LIN {X 0,Y 175.881,Z 377.344,A -85,B 0,C 180,E1 -22792.309,E2 -22792.309} C_VEL
LIN {X 0,Y 178.302,Z 371.488,A -85,B 0,C 180,E1 -22794.961,E2 -22794.961} C_VEL
LIN {X 0,Y 180.637,Z 365.547,A -85,B 0,C 180,E1 -22797.203,E2 -22797.203} C_VEL
LIN {X 0,Y 183.902,Z 356.997,A -85,B 0,C 180,E1 -22799.789,E2 -22799.789} C_VEL
LIN {X 0,Y 186.792,Z 348.822,A -85,B 0,C 180,E1 -22801.786,E2 -22801.786} C_VEL
LIN {X 0,Y 189.518,Z 340.315,A -85,B 0,C 180,E1 -22803.478,E2 -22803.478} C_VEL
LIN {X 0,Y 192.068,Z 331.606,A -85,B 0,C 180,E1 -22804.871,E2 -22804.871} C_VEL
LIN {X 0,Y 194.421,Z 321.851,A -85,B 0,C 180,E1 -22806.133,E2 -22806.133} C_VEL
LIN {X 0,Y 196.471,Z 311.774,A -85,B 0,C 180,E1 -22807.13,E2 -22807.13} C_VEL
LIN {X 0,Y 198.049,Z 301.956,A -85,B 0,C 180,E1 -22807.852,E2 -22807.852} C_VEL
LIN {X 0,Y 199.073,Z 292.344,A -85,B 0,C 180,E1 -22808.374,E2 -22808.374} C_VEL
LIN {X 0,Y 201.449,Z 250.434,A -85,B 0,C 180,E1 -22809.804,E2 -22809.804} C_VEL
LIN {X 0,Y 199.678,Z 238.962,A -85,B 0,C 180,E1 -22810.755,E2 -22810.755} C_VEL
LIN {X 0,Y 194.382,Z 225.961,A -85,B 0,C 180,E1 -22812.741,E2 -22812.741} C_VEL
LIN {X 0,Y 189.399,Z 215.335,A -85,B 0,C 180,E1 -22814.692,E2 -22814.692} C_VEL
LIN {X 0,Y 183.457,Z 204.391,A -85,B 0,C 180,E1 -22817.157,E2 -22817.157} C_VEL
LIN {X 0,Y 180.627,Z 199.673,A -85,B 0,C 180,E1 -22818.402,E2 -22818.402} C_VEL
LIN {X 0,Y 177.944,Z 195.27,A -85,B 0,C 180,E1 -22819.645,E2 -22819.645} C_VEL
LIN {X 0,Y 174.675,Z 190.219,A -85,B 0,C 180,E1 -22821.238,E2 -22821.238} C_VEL
LIN {X 0,Y 172.03,Z 186.816,A -85,B 0,C 180,E1 -22822.576,E2 -22822.576} C_VEL
LIN {X 0,Y 171.463,Z 185.167,A -85,B 0,C 180,E1 -22823.168,E2 -22823.168} C_VEL
LIN {X 0,Y 171.404,Z 184.674,A -85,B 0,C 180,E1 -22823.883,E2 -22823.883} C_VEL
LIN {X 0,Y 171.46,Z 184.628,A -85,B 0,C 180,E1 -22829.403,E2 -22829.403} C_VEL
LIN {X 0,Y 171.463,Z 184.591,A -85,B 0,C 180,E1 -22834.387,E2 -22834.387} C_VEL
LIN {X 0,Y 171.579,Z 184.562,A -85,B 0,C 180,E1 -22840.87,E2 -22840.87} C_VEL
LIN {X 0,Y 171.577,Z 184.609,A -85,B 0,C 180,E1 -22845.772,E2 -22845.772} C_VEL
LIN {X 0,Y 171.848,Z 184.523,A -85,B 0,C 180,E1 -22850.584,E2 -22850.584} C_VEL
LIN {X 0,Y 171.816,Z 184.583,A -85,B 0,C 180,E1 -22855.306,E2 -22855.306} C_VEL
LIN {X 0,Y 172.33,Z 184.463,A -85,B 0,C 180,E1 -22859.999,E2 -22859.999} C_VEL
LIN {X 0,Y 171.822,Z 184.581,A -85,B 0,C 180,E1 -22864.691,E2 -22864.691} C_VEL
LIN {X 0,Y 171.872,Z 184.523,A -85,B 0,C 180,E1 -22869.412,E2 -22869.412} C_VEL
LIN {X 0,Y 171.609,Z 184.608,A -85,B 0,C 180,E1 -22874.223,E2 -22874.223} C_VEL
LIN {X 0,Y 171.542,Z 184.57,A -85,B 0,C 180,E1 -22879.56,E2 -22879.56} C_VEL
LIN {X 0,Y 171.466,Z 184.596,A -85,B 0,C 180,E1 -22885.615,E2 -22885.615} C_VEL
LIN {X 0,Y 171.455,Z 184.624,A -85,B 0,C 180,E1 -22890.595,E2 -22890.595} C_VEL
LIN {X 0,Y 171.407,Z 184.674,A -85,B 0,C 180,E1 -22896.706,E2 -22896.706} C_VEL
LIN {X 0,Y 171.569,Z 185.534,A -85,B 0,C 180,E1 -22897.447,E2 -22897.447} C_VEL
LIN {X 0,Y 173.116,Z 188.45,A -85,B 0,C 180,E1 -22898.383,E2 -22898.383} C_VEL
LIN {X 0,Y 175.17,Z 190.413,A -85,B 0,C 180,E1 -22899.354,E2 -22899.354} C_VEL
LIN {X 0,Y 177.361,Z 193.784,A -85,B 0,C 180,E1 -22900.423,E2 -22900.423} C_VEL
LIN {X 0,Y 178.755,Z 195.514,A -85,B 0,C 180,E1 -22901.052,E2 -22901.052} C_VEL
LIN {X 0,Y 182.889,Z 201.427,A -85,B 0,C 180,E1 -22902.864,E2 -22902.864} C_VEL
LIN {X 0,Y 189.262,Z 210.902,A -85,B 0,C 180,E1 -22905.416,E2 -22905.416} C_VEL
LIN {X 0,Y 196.045,Z 222.621,A -85,B 0,C 180,E1 -22907.921,E2 -22907.921} C_VEL
LIN {X 0,Y 203.07,Z 236.728,A -85,B 0,C 180,E1 -22910.338,E2 -22910.338} C_VEL
LIN {X 0,Y 211.588,Z 254.961,A -85,B 0,C 180,E1 -22913.002,E2 -22913.002} C_VEL
LIN {X 0,Y 220.343,Z 269.518,A -85,B 0,C 180,E1 -22915.279,E2 -22915.279} C_VEL
LIN {X 0,Y 228.476,Z 280.884,A -85,B 0,C 180,E1 -22917.153,E2 -22917.153} C_VEL
LIN {X 0,Y 236.39,Z 290.633,A -85,B 0,C 180,E1 -22918.936,E2 -22918.936} C_VEL
LIN {X 0,Y 244.162,Z 299.37,A -85,B 0,C 180,E1 -22920.704,E2 -22920.704} C_VEL
LIN {X 0,Y 253.056,Z 308.497,A -85,B 0,C 180,E1 -22922.711,E2 -22922.711} C_VEL
LIN {X 0,Y 263.678,Z 317.89,A -85,B 0,C 180,E1 -22924.987,E2 -22924.987} C_VEL
LIN {X 0,Y 276.714,Z 327.934,A -85,B 0,C 180,E1 -22927.606,E2 -22927.606} C_VEL
LIN {X 0,Y 290.97,Z 338.137,A -85,B 0,C 180,E1 -22930.386,E2 -22930.386} C_VEL
LIN {X 0,Y 299.99,Z 344.721,A -85,B 0,C 180,E1 -22932.269,E2 -22932.269} C_VEL
LIN {X 0,Y 305.133,Z 348.259,A -85,B 0,C 180,E1 -22933.436,E2 -22933.436} C_VEL
LIN {X 0,Y 312.318,Z 353.434,A -85,B 0,C 180,E1 -22935.376,E2 -22935.376} C_VEL
LIN {X 0,Y 318.689,Z 357.408,A -85,B 0,C 180,E1 -22937.26,E2 -22937.26} C_VEL
LIN {X 0,Y 322.754,Z 360.096,A -85,B 0,C 180,E1 -22938.698,E2 -22938.698} C_VEL
LIN {X 0,Y 327.517,Z 363.396,A -85,B 0,C 180,E1 -22940.778,E2 -22940.778} C_VEL
LIN {X 0,Y 331.232,Z 365.579,A -85,B 0,C 180,E1 -22942.686,E2 -22942.686} C_VEL
LIN {X 0,Y 333.387,Z 366.65,A -85,B 0,C 180,E1 -22943.95,E2 -22943.95} C_VEL
LIN {X 0,Y 335.126,Z 367.434,A -85,B 0,C 180,E1 -22945.188,E2 -22945.188} C_VEL
LIN {X 0,Y 336.551,Z 367.967,A -85,B 0,C 180,E1 -22946.408,E2 -22946.408} C_VEL
LIN {X 0,Y 337.608,Z 368.387,A -85,B 0,C 180,E1 -22947.714,E2 -22947.714} C_VEL
LIN {X 0,Y 338.327,Z 368.639,A -85,B 0,C 180,E1 -22950,E2 -22950} C_VEL
LIN {X 0,Y 338.048,Z 368.614,A -85,B 0,C 180,E1 -22951.191,E2 -22951.191} C_VEL
LIN {X 0,Y 337.513,Z 368.349,A -85,B 0,C 180,E1 -22952.387,E2 -22952.387} C_VEL
LIN {X 0,Y 336.548,Z 367.946,A -85,B 0,C 180,E1 -22953.592,E2 -22953.592} C_VEL
LIN {X 0,Y 335.116,Z 367.413,A -85,B 0,C 180,E1 -22954.812,E2 -22954.812} C_VEL
LIN {X 0,Y 332.503,Z 366.264,A -85,B 0,C 180,E1 -22956.583,E2 -22956.583} C_VEL
LIN {X 0,Y 328.782,Z 364.143,A -85,B 0,C 180,E1 -22958.605,E2 -22958.605} C_VEL
LIN {X 0,Y 324.587,Z 361.397,A -85,B 0,C 180,E1 -22960.537,E2 -22960.537} C_VEL
LIN {X 0,Y 321.248,Z 359.031,A -85,B 0,C 180,E1 -22961.878,E2 -22961.878} C_VEL
LIN {X 0,Y 317.507,Z 356.675,A -85,B 0,C 180,E1 -22963.114,E2 -22963.114} C_VEL
LIN {X 0,Y 312.317,Z 353.442,A -85,B 0,C 180,E1 -22964.624,E2 -22964.624} C_VEL
LIN {X 0,Y 307.134,Z 349.761,A -85,B 0,C 180,E1 -22966.044,E2 -22966.044} C_VEL
LIN {X 0,Y 301.828,Z 346.015,A -85,B 0,C 180,E1 -22967.319,E2 -22967.319} C_VEL
LIN {X 0,Y 293.694,Z 340.243,A -85,B 0,C 180,E1 -22969.055,E2 -22969.055} C_VEL
LIN {X 0,Y 285.441,Z 334.313,A -85,B 0,C 180,E1 -22970.674,E2 -22970.674} C_VEL
LIN {X 0,Y 272.495,Z 324.875,A -85,B 0,C 180,E1 -22973.216,E2 -22973.216} C_VEL
LIN {X 0,Y 258.338,Z 313.345,A -85,B 0,C 180,E1 -22976.138,E2 -22976.138} C_VEL
LIN {X 0,Y 247.802,Z 303.312,A -85,B 0,C 180,E1 -22978.456,E2 -22978.456} C_VEL
LIN {X 0,Y 238.022,Z 292.543,A -85,B 0,C 180,E1 -22980.689,E2 -22980.689} C_VEL
LIN {X 0,Y 229.51,Z 282.137,A -85,B 0,C 180,E1 -22982.639,E2 -22982.639} C_VEL
LIN {X 0,Y 221.653,Z 271.453,A -85,B 0,C 180,E1 -22984.41,E2 -22984.41} C_VEL
LIN {X 0,Y 212.727,Z 256.998,A -85,B 0,C 180,E1 -22986.681,E2 -22986.681} C_VEL
LIN {X 0,Y 205.697,Z 242.652,A -85,B 0,C 180,E1 -22988.793,E2 -22988.793} C_VEL
LIN {X 0,Y 200.149,Z 230.678,A -85,B 0,C 180,E1 -22990.644,E2 -22990.644} C_VEL
LIN {X 0,Y 193.861,Z 218.632,A -85,B 0,C 180,E1 -22992.866,E2 -22992.866} C_VEL
LIN {X 0,Y 186.678,Z 206.839,A -85,B 0,C 180,E1 -22995.596,E2 -22995.596} C_VEL
LIN {X 0,Y 180.604,Z 198.174,A -85,B 0,C 180,E1 -22998.118,E2 -22998.118} C_VEL
LIN {X 0,Y 177.87,Z 194.262,A -85,B 0,C 180,E1 -22999.355,E2 -22999.355} C_VEL
LIN {X 0,Y 175.623,Z 191.34,A -85,B 0,C 180,E1 -23000.406,E2 -23000.406} C_VEL
LIN {X 0,Y 174.792,Z 189.863,A -85,B 0,C 180,E1 -23000.833,E2 -23000.833} C_VEL
LIN {X 0,Y 172.517,Z 187.642,A -85,B 0,C 180,E1 -23001.924,E2 -23001.924} C_VEL
LIN {X 0,Y 171.488,Z 185.196,A -85,B 0,C 180,E1 -23002.717,E2 -23002.717} C_VEL
LIN {X 0,Y 171.418,Z 184.641,A -85,B 0,C 180,E1 -23003.526,E2 -23003.526} C_VEL
LIN {X 0,Y 171.455,Z 184.624,A -85,B 0,C 180,E1 -23009.405,E2 -23009.405} C_VEL
LIN {X 0,Y 171.466,Z 184.596,A -85,B 0,C 180,E1 -23014.385,E2 -23014.385} C_VEL
LIN {X 0,Y 171.577,Z 184.565,A -85,B 0,C 180,E1 -23020.873,E2 -23020.873} C_VEL
LIN {X 0,Y 171.609,Z 184.608,A -85,B 0,C 180,E1 -23025.777,E2 -23025.777} C_VEL
LIN {X 0,Y 171.872,Z 184.523,A -85,B 0,C 180,E1 -23030.588,E2 -23030.588} C_VEL
LIN {X 0,Y 171.822,Z 184.581,A -85,B 0,C 180,E1 -23035.309,E2 -23035.309} C_VEL
LIN {X 0,Y 172.33,Z 184.463,A -85,B 0,C 180,E1 -23040.001,E2 -23040.001} C_VEL
LIN {X 0,Y 171.816,Z 184.583,A -85,B 0,C 180,E1 -23044.694,E2 -23044.694} C_VEL
LIN {X 0,Y 171.848,Z 184.523,A -85,B 0,C 180,E1 -23049.416,E2 -23049.416} C_VEL
LIN {X 0,Y 171.577,Z 184.609,A -85,B 0,C 180,E1 -23054.228,E2 -23054.228} C_VEL
LIN {X 0,Y 171.545,Z 184.568,A -85,B 0,C 180,E1 -23059.563,E2 -23059.563} C_VEL
LIN {X 0,Y 171.463,Z 184.591,A -85,B 0,C 180,E1 -23065.613,E2 -23065.613} C_VEL
LIN {X 0,Y 171.46,Z 184.628,A -85,B 0,C 180,E1 -23070.597,E2 -23070.597} C_VEL
LIN {X 0,Y 171.404,Z 184.741,A -85,B 0,C 180,E1 -23076.39,E2 -23076.39} C_VEL
LIN {X 0,Y 171.537,Z 185.46,A -85,B 0,C 180,E1 -23076.998,E2 -23076.998} C_VEL
LIN {X 0,Y 173.002,Z 188.32,A -85,B 0,C 180,E1 -23077.947,E2 -23077.947} C_VEL
LIN {X 0,Y 175.535,Z 191.428,A -85,B 0,C 180,E1 -23079.185,E2 -23079.185} C_VEL
LIN {X 0,Y 178.482,Z 195.95,A -85,B 0,C 180,E1 -23080.598,E2 -23080.598} C_VEL
LIN {X 0,Y 184.372,Z 205.931,A -85,B 0,C 180,E1 -23083.233,E2 -23083.233} C_VEL
LIN {X 0,Y 191.12,Z 218.728,A -85,B 0,C 180,E1 -23085.987,E2 -23085.987} C_VEL
LIN {X 0,Y 196.979,Z 232.036,A -85,B 0,C 180,E1 -23088.239,E2 -23088.239} C_VEL
LIN {X 0,Y 199.946,Z 239.938,A -85,B 0,C 180,E1 -23089.355,E2 -23089.355} C_VEL
LIN {X 0,Y 201.455,Z 251.296,A -85,B 0,C 180,E1 -23090.237,E2 -23090.237} C_VEL
LIN {X 0,Y 199.128,Z 292.429,A -85,B 0,C 180,E1 -23091.639,E2 -23091.639} C_VEL
LIN {X 0,Y 197.838,Z 303.708,A -85,B 0,C 180,E1 -23092.262,E2 -23092.262} C_VEL
LIN {X 0,Y 195.577,Z 316.798,A -85,B 0,C 180,E1 -23093.315,E2 -23093.315} C_VEL
LIN {X 0,Y 192.881,Z 328.342,A -85,B 0,C 180,E1 -23094.66,E2 -23094.66} C_VEL
LIN {X 0,Y 190.404,Z 337.616,A -85,B 0,C 180,E1 -23096.064,E2 -23096.064} C_VEL
LIN {X 0,Y 187.564,Z 346.555,A -85,B 0,C 180,E1 -23097.728,E2 -23097.728} C_VEL
LIN {X 0,Y 184.594,Z 355.079,A -85,B 0,C 180,E1 -23099.705,E2 -23099.705} C_VEL
LIN {X 0,Y 181.875,Z 362.294,A -85,B 0,C 180,E1 -23101.747,E2 -23101.747} C_VEL
LIN {X 0,Y 179.441,Z 368.494,A -85,B 0,C 180,E1 -23103.857,E2 -23103.857} C_VEL
LIN {X 0,Y 176.891,Z 375.034,A -85,B 0,C 180,E1 -23106.59,E2 -23106.59} C_VEL
LIN {X 0,Y 174.916,Z 379.533,A -85,B 0,C 180,E1 -23108.801,E2 -23108.801} C_VEL
LIN {X 0,Y 172.575,Z 385.026,A -85,B 0,C 180,E1 -23112.216,E2 -23112.216} C_VEL
LIN {X 0,Y 170.804,Z 389.353,A -85,B 0,C 180,E1 -23115.707,E2 -23115.707} C_VEL
LIN {X 0,Y 170.014,Z 391.725,A -85,B 0,C 180,E1 -23118.072,E2 -23118.072} C_VEL
LIN {X 0,Y 169.417,Z 393.528,A -85,B 0,C 180,E1 -23120.449,E2 -23120.449} C_VEL
LIN {X 0,Y 168.933,Z 395.987,A -85,B 0,C 180,E1 -23125.227,E2 -23125.227} C_VEL
LIN {X 0,Y 168.87,Z 396.632,A -85,B 0,C 180,E1 -23128.403,E2 -23128.403} C_VEL
LIN {X 0,Y 168.968,Z 396.739,A -85,B 0,C 180,E1 -23130,E2 -23130} C_VEL
LIN {X 0,Y 168.853,Z 396.52,A -85,B 0,C 180,E1 -23132.627,E2 -23132.627} C_VEL
LIN {X 0,Y 168.863,Z 395.985,A -85,B 0,C 180,E1 -23134.775,E2 -23134.775} C_VEL
LIN {X 0,Y 169.206,Z 394.079,A -85,B 0,C 180,E1 -23138.609,E2 -23138.609} C_VEL
LIN {X 0,Y 168.94,Z 392.807,A -85,B 0,C 180,E1 -23140.562,E2 -23140.562} C_VEL
LIN {X 0,Y 167.039,Z 390.176,A -85,B 0,C 180,E1 -23143.759,E2 -23143.759} C_VEL
LIN {X 0,Y 165.574,Z 386.861,A -85,B 0,C 180,E1 -23146.944,E2 -23146.944} C_VEL
LIN {X 0,Y 165.991,Z 384.451,A -85,B 0,C 180,E1 -23148.809,E2 -23148.809} C_VEL
LIN {X 0,Y 168.795,Z 378.306,A -85,B 0,C 180,E1 -23152.652,E2 -23152.652} C_VEL
LIN {X 0,Y 171.612,Z 371.914,A -85,B 0,C 180,E1 -23155.712,E2 -23155.712} C_VEL
LIN {X 0,Y 174.324,Z 365.355,A -85,B 0,C 180,E1 -23158.275,E2 -23158.275} C_VEL
LIN {X 0,Y 177.77,Z 356.805,A -85,B 0,C 180,E1 -23160.927,E2 -23160.927} C_VEL
LIN {X 0,Y 180.789,Z 348.631,A -85,B 0,C 180,E1 -23162.972,E2 -23162.972} C_VEL
LIN {X 0,Y 183.635,Z 340.123,A -85,B 0,C 180,E1 -23164.7,E2 -23164.7} C_VEL
LIN {X 0,Y 186.275,Z 331.414,A -85,B 0,C 180,E1 -23166.122,E2 -23166.122} C_VEL
LIN {X 0,Y 188.748,Z 321.66,A -85,B 0,C 180,E1 -23167.401,E2 -23167.401} C_VEL
LIN {X 0,Y 190.873,Z 311.583,A -85,B 0,C 180,E1 -23168.414,E2 -23168.414} C_VEL
LIN {X 0,Y 192.584,Z 301.13,A -85,B 0,C 180,E1 -23169.188,E2 -23169.188} C_VEL
LIN {X 0,Y 193.649,Z 291.081,A -85,B 0,C 180,E1 -23169.724,E2 -23169.724} C_VEL
LIN {X 0,Y 195.927,Z 251.075,A -85,B 0,C 180,E1 -23171.123,E2 -23171.123} C_VEL
LIN {X 0,Y 194.532,Z 241.871,A -85,B 0,C 180,E1 -23171.925,E2 -23171.925} C_VEL
LIN {X 0,Y 189.455,Z 229.158,A -85,B 0,C 180,E1 -23173.96,E2 -23173.96} C_VEL
LIN {X 0,Y 184.476,Z 218.447,A -85,B 0,C 180,E1 -23176.044,E2 -23176.044} C_VEL
LIN {X 0,Y 177.787,Z 206.032,A -85,B 0,C 180,E1 -23179.053,E2 -23179.053} C_VEL
LIN {X 0,Y 174.086,Z 200.115,A -85,B 0,C 180,E1 -23180.843,E2 -23180.843} C_VEL
LIN {X 0,Y 171.293,Z 195.651,A -85,B 0,C 180,E1 -23182.294,E2 -23182.294} C_VEL
LIN {X 0,Y 168.602,Z 191.975,A -85,B 0,C 180,E1 -23183.743,E2 -23183.743} C_VEL
LIN {X 0,Y 167.935,Z 190.842,A -85,B 0,C 180,E1 -23184.132,E2 -23184.132} C_VEL
LIN {X 0,Y 165.524,Z 188.584,A -85,B 0,C 180,E1 -23185.463,E2 -23185.463} C_VEL
LIN {X 0,Y 164.436,Z 186.081,A -85,B 0,C 180,E1 -23186.42,E2 -23186.42} C_VEL
LIN {X 0,Y 164.372,Z 185.526,A -85,B 0,C 180,E1 -23187.272,E2 -23187.272} C_VEL
LIN {X 0,Y 164.341,Z 185.476,A -85,B 0,C 180,E1 -23191.938,E2 -23191.938} C_VEL
LIN {X 0,Y 164.411,Z 185.471,A -85,B 0,C 180,E1 -23194.692,E2 -23194.692} C_VEL
LIN {X 0,Y 164.485,Z 185.449,A -85,B 0,C 180,E1 -23200.05,E2 -23200.05} C_VEL
LIN {X 0,Y 164.524,Z 185.484,A -85,B 0,C 180,E1 -23205.148,E2 -23205.148} C_VEL
LIN {X 0,Y 164.767,Z 185.404,A -85,B 0,C 180,E1 -23210.175,E2 -23210.175} C_VEL
LIN {X 0,Y 164.831,Z 185.413,A -85,B 0,C 180,E1 -23212.65,E2 -23212.65} C_VEL
LIN {X 0,Y 165.047,Z 185.39,A -85,B 0,C 180,E1 -23217.558,E2 -23217.558} C_VEL
LIN {X 0,Y 165.292,Z 185.339,A -85,B 0,C 180,E1 -23219.999,E2 -23219.999} C_VEL
LIN {X 0,Y 164.772,Z 185.461,A -85,B 0,C 180,E1 -23224.892,E2 -23224.892} C_VEL
LIN {X 0,Y 164.846,Z 185.416,A -85,B 0,C 180,E1 -23227.347,E2 -23227.347} C_VEL
LIN {X 0,Y 164.749,Z 185.414,A -85,B 0,C 180,E1 -23231.145,E2 -23231.145} C_VEL
LIN {X 0,Y 164.502,Z 185.454,A -85,B 0,C 180,E1 -23237.4,E2 -23237.4} C_VEL
LIN {X 0,Y 164.471,Z 185.452,A -85,B 0,C 180,E1 -23239.988,E2 -23239.988} C_VEL
LIN {X 0,Y 164.391,Z 185.472,A -85,B 0,C 180,E1 -23246.133,E2 -23246.133} C_VEL
LIN {X 0,Y 164.385,Z 185.491,A -85,B 0,C 180,E1 -23252.377,E2 -23252.377} C_VEL
LIN {X 0,Y 164.377,Z 185.815,A -85,B 0,C 180,E1 -23253.766,E2 -23253.766} C_VEL
LIN {X 0,Y 164.763,Z 187.147,A -85,B 0,C 180,E1 -23254.405,E2 -23254.405} C_VEL
LIN {X 0,Y 166.409,Z 189.67,A -85,B 0,C 180,E1 -23255.434,E2 -23255.434} C_VEL
LIN {X 0,Y 168.275,Z 191.164,A -85,B 0,C 180,E1 -23256.429,E2 -23256.429} C_VEL
LIN {X 0,Y 170.195,Z 194.383,A -85,B 0,C 180,E1 -23257.522,E2 -23257.522} C_VEL
LIN {X 0,Y 172.038,Z 196.358,A -85,B 0,C 180,E1 -23258.45,E2 -23258.45} C_VEL
LIN {X 0,Y 174.59,Z 199.966,A -85,B 0,C 180,E1 -23259.729,E2 -23259.729} C_VEL
LIN {X 0,Y 180.932,Z 209.13,A -85,B 0,C 180,E1 -23262.634,E2 -23262.634} C_VEL
LIN {X 0,Y 186.915,Z 218.677,A -85,B 0,C 180,E1 -23265.113,E2 -23265.113} C_VEL
LIN {X 0,Y 192.735,Z 229.168,A -85,B 0,C 180,E1 -23267.347,E2 -23267.347} C_VEL
LIN {X 0,Y 199.084,Z 242.459,A -85,B 0,C 180,E1 -23269.641,E2 -23269.641} C_VEL
LIN {X 0,Y 206.912,Z 259.443,A -85,B 0,C 180,E1 -23272.207,E2 -23272.207} C_VEL
LIN {X 0,Y 215.763,Z 274.325,A -85,B 0,C 180,E1 -23274.619,E2 -23274.619} C_VEL
LIN {X 0,Y 223.821,Z 285.817,A -85,B 0,C 180,E1 -23276.619,E2 -23276.619} C_VEL
LIN {X 0,Y 233.409,Z 297.849,A -85,B 0,C 180,E1 -23279.043,E2 -23279.043} C_VEL
LIN {X 0,Y 242.631,Z 308.097,A -85,B 0,C 180,E1 -23281.355,E2 -23281.355} C_VEL
LIN {X 0,Y 252.683,Z 317.792,A -85,B 0,C 180,E1 -23283.762,E2 -23283.762} C_VEL
LIN {X 0,Y 265.457,Z 328.251,A -85,B 0,C 180,E1 -23286.602,E2 -23286.602} C_VEL
LIN {X 0,Y 278.514,Z 337.618,A -85,B 0,C 180,E1 -23289.312,E2 -23289.312} C_VEL
LIN {X 0,Y 289.061,Z 344.904,A -85,B 0,C 180,E1 -23291.478,E2 -23291.478} C_VEL
LIN {X 0,Y 298.801,Z 351.715,A -85,B 0,C 180,E1 -23293.606,E2 -23293.606} C_VEL
LIN {X 0,Y 305.375,Z 356.469,A -85,B 0,C 180,E1 -23295.336,E2 -23295.336} C_VEL
LIN {X 0,Y 310.985,Z 360.104,A -85,B 0,C 180,E1 -23296.939,E2 -23296.939} C_VEL
LIN {X 0,Y 315.669,Z 362.977,A -85,B 0,C 180,E1 -23298.441,E2 -23298.441} C_VEL
LIN {X 0,Y 320.632,Z 366.467,A -85,B 0,C 180,E1 -23300.522,E2 -23300.522} C_VEL
LIN {X 0,Y 325.665,Z 369.51,A -85,B 0,C 180,E1 -23303.067,E2 -23303.067} C_VEL
LIN {X 0,Y 328.828,Z 371.056,A -85,B 0,C 180,E1 -23305.096,E2 -23305.096} C_VEL
LIN {X 0,Y 330.816,Z 371.833,A -85,B 0,C 180,E1 -23306.833,E2 -23306.833} C_VEL
LIN {X 0,Y 331.953,Z 372.324,A -85,B 0,C 180,E1 -23308.787,E2 -23308.787} C_VEL
LIN {X 0,Y 332.278,Z 372.333,A -85,B 0,C 180,E1 -23310,E2 -23310} C_VEL
LIN {X 0,Y 331.969,Z 372.307,A -85,B 0,C 180,E1 -23311.213,E2 -23311.213} C_VEL
LIN {X 0,Y 330.821,Z 371.835,A -85,B 0,C 180,E1 -23313.181,E2 -23313.181} C_VEL
LIN {X 0,Y 328.814,Z 371.044,A -85,B 0,C 180,E1 -23314.904,E2 -23314.904} C_VEL
LIN {X 0,Y 325.665,Z 369.505,A -85,B 0,C 180,E1 -23316.933,E2 -23316.933} C_VEL
LIN {X 0,Y 322.114,Z 367.424,A -85,B 0,C 180,E1 -23318.785,E2 -23318.785} C_VEL
LIN {X 0,Y 319.119,Z 365.447,A -85,B 0,C 180,E1 -23320.148,E2 -23320.148} C_VEL
LIN {X 0,Y 315.63,Z 363.006,A -85,B 0,C 180,E1 -23321.56,E2 -23321.56} C_VEL
LIN {X 0,Y 310.431,Z 359.762,A -85,B 0,C 180,E1 -23323.224,E2 -23323.224} C_VEL
LIN {X 0,Y 305.19,Z 356.343,A -85,B 0,C 180,E1 -23324.722,E2 -23324.722} C_VEL
LIN {X 0,Y 298.734,Z 351.703,A -85,B 0,C 180,E1 -23326.398,E2 -23326.398} C_VEL
LIN {X 0,Y 291.766,Z 346.896,A -85,B 0,C 180,E1 -23327.929,E2 -23327.929} C_VEL
LIN {X 0,Y 283.598,Z 341.056,A -85,B 0,C 180,E1 -23329.664,E2 -23329.664} C_VEL
LIN {X 0,Y 269.955,Z 331.548,A -85,B 0,C 180,E1 -23332.454,E2 -23332.454} C_VEL
LIN {X 0,Y 256.61,Z 321.192,A -85,B 0,C 180,E1 -23335.34,E2 -23335.34} C_VEL
LIN {X 0,Y 246.207,Z 311.766,A -85,B 0,C 180,E1 -23337.763,E2 -23337.763} C_VEL
LIN {X 0,Y 236.022,Z 300.893,A -85,B 0,C 180,E1 -23340.287,E2 -23340.287} C_VEL
LIN {X 0,Y 227.311,Z 290.369,A -85,B 0,C 180,E1 -23342.493,E2 -23342.493} C_VEL
LIN {X 0,Y 219.314,Z 279.593,A -85,B 0,C 180,E1 -23344.498,E2 -23344.498} C_VEL
LIN {X 0,Y 210.189,Z 265.266,A -85,B 0,C 180,E1 -23346.855,E2 -23346.855} C_VEL
LIN {X 0,Y 202.831,Z 251.158,A -85,B 0,C 180,E1 -23349.069,E2 -23349.069} C_VEL
LIN {X 0,Y 196.148,Z 236.12,A -85,B 0,C 180,E1 -23351.401,E2 -23351.401} C_VEL
LIN {X 0,Y 189.843,Z 223.734,A -85,B 0,C 180,E1 -23353.746,E2 -23353.746} C_VEL
LIN {X 0,Y 182.773,Z 211.915,A -85,B 0,C 180,E1 -23356.583,E2 -23356.583} C_VEL
LIN {X 0,Y 176.942,Z 203.408,A -85,B 0,C 180,E1 -23359.147,E2 -23359.147} C_VEL
LIN {X 0,Y 174.22,Z 199.577,A -85,B 0,C 180,E1 -23360.444,E2 -23360.444} C_VEL
LIN {X 0,Y 171.417,Z 195.571,A -85,B 0,C 180,E1 -23361.867,E2 -23361.867} C_VEL
LIN {X 0,Y 169.147,Z 192.916,A -85,B 0,C 180,E1 -23363.048,E2 -23363.048} C_VEL
LIN {X 0,Y 167.92,Z 190.819,A -85,B 0,C 180,E1 -23363.761,E2 -23363.761} C_VEL
LIN {X 0,Y 165.693,Z 188.828,A -85,B 0,C 180,E1 -23364.981,E2 -23364.981} C_VEL
LIN {X 0,Y 164.426,Z 186.04,A -85,B 0,C 180,E1 -23366.038,E2 -23366.038} C_VEL
LIN {X 0,Y 164.345,Z 185.511,A -85,B 0,C 180,E1 -23366.923,E2 -23366.923} C_VEL
LIN {X 0,Y 164.402,Z 185.506,A -85,B 0,C 180,E1 -23369.139,E2 -23369.139} C_VEL
LIN {X 0,Y 164.414,Z 185.477,A -85,B 0,C 180,E1 -23374.695,E2 -23374.695} C_VEL
LIN {X 0,Y 164.483,Z 185.45,A -85,B 0,C 180,E1 -23380.052,E2 -23380.052} C_VEL
LIN {X 0,Y 164.552,Z 185.488,A -85,B 0,C 180,E1 -23385.153,E2 -23385.153} C_VEL
LIN {X 0,Y 164.796,Z 185.403,A -85,B 0,C 180,E1 -23390.179,E2 -23390.179} C_VEL
LIN {X 0,Y 164.846,Z 185.416,A -85,B 0,C 180,E1 -23392.653,E2 -23392.653} C_VEL
LIN {X 0,Y 165.049,Z 185.385,A -85,B 0,C 180,E1 -23397.561,E2 -23397.561} C_VEL
LIN {X 0,Y 165.292,Z 185.339,A -85,B 0,C 180,E1 -23400.001,E2 -23400.001} C_VEL
LIN {X 0,Y 164.765,Z 185.462,A -85,B 0,C 180,E1 -23404.895,E2 -23404.895} C_VEL
LIN {X 0,Y 164.831,Z 185.413,A -85,B 0,C 180,E1 -23407.35,E2 -23407.35} C_VEL
LIN {X 0,Y 164.703,Z 185.419,A -85,B 0,C 180,E1 -23411.062,E2 -23411.062} C_VEL
LIN {X 0,Y 164.524,Z 185.484,A -85,B 0,C 180,E1 -23414.852,E2 -23414.852} C_VEL
LIN {X 0,Y 164.474,Z 185.451,A -85,B 0,C 180,E1 -23419.99,E2 -23419.99} C_VEL
LIN {X 0,Y 164.389,Z 185.468,A -85,B 0,C 180,E1 -23426.131,E2 -23426.131} C_VEL
LIN {X 0,Y 164.388,Z 185.5,A -85,B 0,C 180,E1 -23432.38,E2 -23432.38} C_VEL
LIN {X 0,Y 164.407,Z 185.864,A -85,B 0,C 180,E1 -23433.413,E2 -23433.413} C_VEL
LIN {X 0,Y 164.775,Z 187.218,A -85,B 0,C 180,E1 -23434.039,E2 -23434.039} C_VEL
LIN {X 0,Y 166.481,Z 189.733,A -85,B 0,C 180,E1 -23435.093,E2 -23435.093} C_VEL
LIN {X 0,Y 168.279,Z 191.289,A -85,B 0,C 180,E1 -23436.06,E2 -23436.06} C_VEL
LIN {X 0,Y 170.328,Z 194.545,A -85,B 0,C 180,E1 -23437.212,E2 -23437.212} C_VEL
LIN {X 0,Y 172.255,Z 197.096,A -85,B 0,C 180,E1 -23438.21,E2 -23438.21} C_VEL
LIN {X 0,Y 176.099,Z 203.374,A -85,B 0,C 180,E1 -23440.151,E2 -23440.151} C_VEL
LIN {X 0,Y 180.309,Z 210.544,A -85,B 0,C 180,E1 -23442.119,E2 -23442.119} C_VEL
LIN {X 0,Y 186.583,Z 222.723,A -85,B 0,C 180,E1 -23444.847,E2 -23444.847} C_VEL
LIN {X 0,Y 192.394,Z 236.231,A -85,B 0,C 180,E1 -23447.225,E2 -23447.225} C_VEL
LIN {X 0,Y 194.779,Z 242.867,A -85,B 0,C 180,E1 -23448.188,E2 -23448.188} C_VEL
LIN {X 0,Y 195.973,Z 251.524,A -85,B 0,C 180,E1 -23448.91,E2 -23448.91} C_VEL
LIN {X 0,Y 193.632,Z 292.079,A -85,B 0,C 180,E1 -23450.329,E2 -23450.329} C_VEL
LIN {X 0,Y 192.31,Z 303.337,A -85,B 0,C 180,E1 -23450.958,E2 -23450.958} C_VEL
LIN {X 0,Y 189.933,Z 316.607,A -85,B 0,C 180,E1 -23452.036,E2 -23452.036} C_VEL
LIN {X 0,Y 187.139,Z 328.151,A -85,B 0,C 180,E1 -23453.403,E2 -23453.403} C_VEL
LIN {X 0,Y 184.554,Z 337.424,A -85,B 0,C 180,E1 -23454.833,E2 -23454.833} C_VEL
LIN {X 0,Y 181.606,Z 346.363,A -85,B 0,C 180,E1 -23456.533,E2 -23456.533} C_VEL
LIN {X 0,Y 178.471,Z 354.886,A -85,B 0,C 180,E1 -23458.549,E2 -23458.549} C_VEL
LIN {X 0,Y 175.63,Z 362.102,A -85,B 0,C 180,E1 -23460.647,E2 -23460.647} C_VEL
LIN {X 0,Y 173.072,Z 368.302,A -85,B 0,C 180,E1 -23462.817,E2 -23462.817} C_VEL
LIN {X 0,Y 170.358,Z 374.842,A -85,B 0,C 180,E1 -23465.636,E2 -23465.636} C_VEL
LIN {X 0,Y 168.289,Z 379.341,A -85,B 0,C 180,E1 -23467.923,E2 -23467.923} C_VEL
LIN {X 0,Y 165.816,Z 384.834,A -85,B 0,C 180,E1 -23471.465,E2 -23471.465} C_VEL
LIN {X 0,Y 163.883,Z 389.16,A -85,B 0,C 180,E1 -23475.09,E2 -23475.09} C_VEL
LIN {X 0,Y 163.041,Z 391.532,A -85,B 0,C 180,E1 -23477.554,E2 -23477.554} C_VEL
LIN {X 0,Y 162.398,Z 393.336,A -85,B 0,C 180,E1 -23480.032,E2 -23480.032} C_VEL
LIN {X 0,Y 161.851,Z 395.795,A -85,B 0,C 180,E1 -23485.018,E2 -23485.018} C_VEL
LIN {X 0,Y 161.8,Z 396.389,A -85,B 0,C 180,E1 -23487.511,E2 -23487.511} C_VEL
LIN {X 0,Y 161.884,Z 396.548,A -85,B 0,C 180,E1 -23490,E2 -23490} C_VEL
LIN {X 0,Y 161.763,Z 396.388,A -85,B 0,C 180,E1 -23492.49,E2 -23492.49} C_VEL
LIN {X 0,Y 161.766,Z 395.793,A -85,B 0,C 180,E1 -23494.985,E2 -23494.985} C_VEL
LIN {X 0,Y 162.376,Z 393.335,A -85,B 0,C 180,E1 -23499.97,E2 -23499.97} C_VEL
LIN {X 0,Y 163.427,Z 390.379,A -85,B 0,C 180,E1 -23503.681,E2 -23503.681} C_VEL
LIN {X 0,Y 165.06,Z 386.386,A -85,B 0,C 180,E1 -23507.34,E2 -23507.34} C_VEL
LIN {X 0,Y 165.991,Z 384.451,A -85,B 0,C 180,E1 -23508.809,E2 -23508.809} C_VEL
LIN {X 0,Y 166.55,Z 381.856,A -85,B 0,C 180,E1 -23510.628,E2 -23510.628} C_VEL
LIN {X 0,Y 165.958,Z 377.196,A -85,B 0,C 180,E1 -23513.641,E2 -23513.641} C_VEL
LIN {X 0,Y 165.647,Z 372.04,A -85,B 0,C 180,E1 -23516.561,E2 -23516.561} C_VEL
LIN {X 0,Y 166.623,Z 368.424,A -85,B 0,C 180,E1 -23518.171,E2 -23518.171} C_VEL
LIN {X 0,Y 170.197,Z 360.284,A -85,B 0,C 180,E1 -23521.075,E2 -23521.075} C_VEL
LIN {X 0,Y 174.458,Z 349.573,A -85,B 0,C 180,E1 -23523.983,E2 -23523.983} C_VEL
LIN {X 0,Y 177.406,Z 341.283,A -85,B 0,C 180,E1 -23525.755,E2 -23525.755} C_VEL
LIN {X 0,Y 180.585,Z 331.222,A -85,B 0,C 180,E1 -23527.451,E2 -23527.451} C_VEL
LIN {X 0,Y 183.169,Z 321.469,A -85,B 0,C 180,E1 -23528.747,E2 -23528.747} C_VEL
LIN {X 0,Y 185.377,Z 311.392,A -85,B 0,C 180,E1 -23529.774,E2 -23529.774} C_VEL
LIN {X 0,Y 187.128,Z 300.987,A -85,B 0,C 180,E1 -23530.559,E2 -23530.559} C_VEL
LIN {X 0,Y 188.161,Z 291.748,A -85,B 0,C 180,E1 -23531.07,E2 -23531.07} C_VEL
LIN {X 0,Y 190.581,Z 252.189,A -85,B 0,C 180,E1 -23532.477,E2 -23532.477} C_VEL
LIN {X 0,Y 189.432,Z 244.667,A -85,B 0,C 180,E1 -23533.174,E2 -23533.174} C_VEL
LIN {X 0,Y 184.522,Z 232.205,A -85,B 0,C 180,E1 -23535.281,E2 -23535.281} C_VEL
LIN {X 0,Y 179.89,Z 222.208,A -85,B 0,C 180,E1 -23537.353,E2 -23537.353} C_VEL
LIN {X 0,Y 174.009,Z 211.003,A -85,B 0,C 180,E1 -23540.184,E2 -23540.184} C_VEL
LIN {X 0,Y 170.266,Z 204.841,A -85,B 0,C 180,E1 -23542.12,E2 -23542.12} C_VEL
LIN {X 0,Y 167.846,Z 200.943,A -85,B 0,C 180,E1 -23543.46,E2 -23543.46} C_VEL
LIN {X 0,Y 164.841,Z 196.752,A -85,B 0,C 180,E1 -23545.194,E2 -23545.194} C_VEL
LIN {X 0,Y 162.358,Z 193.942,A -85,B 0,C 180,E1 -23546.686,E2 -23546.686} C_VEL
LIN {X 0,Y 161.138,Z 191.822,A -85,B 0,C 180,E1 -23547.518,E2 -23547.518} C_VEL
LIN {X 0,Y 158.706,Z 189.741,A -85,B 0,C 180,E1 -23549.092,E2 -23549.092} C_VEL
LIN {X 0,Y 157.381,Z 186.949,A -85,B 0,C 180,E1 -23550.394,E2 -23550.394} C_VEL
LIN {X 0,Y 157.297,Z 186.405,A -85,B 0,C 180,E1 -23551.294,E2 -23551.294} C_VEL
LIN {X 0,Y 157.311,Z 186.378,A -85,B 0,C 180,E1 -23556.29,E2 -23556.29} C_VEL
LIN {X 0,Y 157.409,Z 186.325,A -85,B 0,C 180,E1 -23561.786,E2 -23561.786} C_VEL
LIN {X 0,Y 157.529,Z 186.336,A -85,B 0,C 180,E1 -23567.109,E2 -23567.109} C_VEL
LIN {X 0,Y 157.689,Z 186.286,A -85,B 0,C 180,E1 -23569.729,E2 -23569.729} C_VEL
LIN {X 0,Y 157.767,Z 186.287,A -85,B 0,C 180,E1 -23572.319,E2 -23572.319} C_VEL
LIN {X 0,Y 158.255,Z 186.214,A -85,B 0,C 180,E1 -23579.999,E2 -23579.999} C_VEL
LIN {X 0,Y 157.784,Z 186.29,A -85,B 0,C 180,E1 -23587.678,E2 -23587.678} C_VEL
LIN {X 0,Y 157.679,Z 186.294,A -85,B 0,C 180,E1 -23591.315,E2 -23591.315} C_VEL
LIN {X 0,Y 157.476,Z 186.357,A -85,B 0,C 180,E1 -23595.53,E2 -23595.53} C_VEL
LIN {X 0,Y 157.368,Z 186.344,A -85,B 0,C 180,E1 -23600.932,E2 -23600.932} C_VEL
LIN {X 0,Y 157.311,Z 186.35,A -85,B 0,C 180,E1 -23606.683,E2 -23606.683} C_VEL
LIN {X 0,Y 157.328,Z 186.674,A -85,B 0,C 180,E1 -23609.706,E2 -23609.706} C_VEL
LIN {X 0,Y 157.673,Z 187.862,A -85,B 0,C 180,E1 -23610.464,E2 -23610.464} C_VEL
LIN {X 0,Y 159.203,Z 190.362,A -85,B 0,C 180,E1 -23611.635,E2 -23611.635} C_VEL
LIN {X 0,Y 161.451,Z 192.096,A -85,B 0,C 180,E1 -23613.056,E2 -23613.056} C_VEL
LIN {X 0,Y 163.477,Z 195.455,A -85,B 0,C 180,E1 -23614.397,E2 -23614.397} C_VEL
LIN {X 0,Y 165.509,Z 197.573,A -85,B 0,C 180,E1 -23615.574,E2 -23615.574} C_VEL
LIN {X 0,Y 168.076,Z 201.156,A -85,B 0,C 180,E1 -23617.039,E2 -23617.039} C_VEL
LIN {X 0,Y 169.597,Z 203.288,A -85,B 0,C 180,E1 -23617.865,E2 -23617.865} C_VEL
LIN {X 0,Y 172.697,Z 207.657,A -85,B 0,C 180,E1 -23619.459,E2 -23619.459} C_VEL
LIN {X 0,Y 178.249,Z 215.949,A -85,B 0,C 180,E1 -23622.086,E2 -23622.086} C_VEL
LIN {X 0,Y 183.591,Z 224.799,A -85,B 0,C 180,E1 -23624.401,E2 -23624.401} C_VEL
LIN {X 0,Y 188.923,Z 234.749,A -85,B 0,C 180,E1 -23626.553,E2 -23626.553} C_VEL
LIN {X 0,Y 194.587,Z 247.049,A -85,B 0,C 180,E1 -23628.719,E2 -23628.719} C_VEL
LIN {X 0,Y 202.23,Z 263.839,A -85,B 0,C 180,E1 -23631.36,E2 -23631.36} C_VEL
LIN {X 0,Y 211.13,Z 279.041,A -85,B 0,C 180,E1 -23633.925,E2 -23633.925} C_VEL
LIN {X 0,Y 218.118,Z 289.426,A -85,B 0,C 180,E1 -23635.859,E2 -23635.859} C_VEL
LIN {X 0,Y 226.087,Z 299.905,A -85,B 0,C 180,E1 -23638.099,E2 -23638.099} C_VEL
LIN {X 0,Y 234.41,Z 309.57,A -85,B 0,C 180,E1 -23640.395,E2 -23640.395} C_VEL
LIN {X 0,Y 242.758,Z 318.279,A -85,B 0,C 180,E1 -23642.627,E2 -23642.627} C_VEL
LIN {X 0,Y 253.559,Z 327.7,A -85,B 0,C 180,E1 -23645.289,E2 -23645.289} C_VEL
LIN {X 0,Y 265.342,Z 336.567,A -85,B 0,C 180,E1 -23647.974,E2 -23647.974} C_VEL
LIN {X 0,Y 278.84,Z 345.674,A -85,B 0,C 180,E1 -23650.874,E2 -23650.874} C_VEL
LIN {X 0,Y 289.824,Z 353.121,A -85,B 0,C 180,E1 -23653.298,E2 -23653.298} C_VEL
LIN {X 0,Y 296.496,Z 357.754,A -85,B 0,C 180,E1 -23654.886,E2 -23654.886} C_VEL
LIN {X 0,Y 303.243,Z 362.435,A -85,B 0,C 180,E1 -23656.751,E2 -23656.751} C_VEL
LIN {X 0,Y 309.772,Z 366.471,A -85,B 0,C 180,E1 -23658.783,E2 -23658.783} C_VEL
LIN {X 0,Y 313.637,Z 369.208,A -85,B 0,C 180,E1 -23660.381,E2 -23660.381} C_VEL
LIN {X 0,Y 318.724,Z 372.421,A -85,B 0,C 180,E1 -23662.864,E2 -23662.864} C_VEL
LIN {X 0,Y 322.199,Z 374.133,A -85,B 0,C 180,E1 -23664.995,E2 -23664.995} C_VEL
LIN {X 0,Y 323.942,Z 374.862,A -85,B 0,C 180,E1 -23666.347,E2 -23666.347} C_VEL
LIN {X 0,Y 325.003,Z 375.291,A -85,B 0,C 180,E1 -23667.521,E2 -23667.521} C_VEL
LIN {X 0,Y 325.633,Z 375.574,A -85,B 0,C 180,E1 -23668.763,E2 -23668.763} C_VEL
LIN {X 0,Y 325.966,Z 375.601,A -85,B 0,C 180,E1 -23670,E2 -23670} C_VEL
LIN {X 0,Y 325.644,Z 375.562,A -85,B 0,C 180,E1 -23671.237,E2 -23671.237} C_VEL
LIN {X 0,Y 325.008,Z 375.279,A -85,B 0,C 180,E1 -23672.479,E2 -23672.479} C_VEL
LIN {X 0,Y 323.83,Z 374.817,A -85,B 0,C 180,E1 -23673.733,E2 -23673.733} C_VEL
LIN {X 0,Y 322.187,Z 374.133,A -85,B 0,C 180,E1 -23675.006,E2 -23675.006} C_VEL
LIN {X 0,Y 318.725,Z 372.388,A -85,B 0,C 180,E1 -23677.137,E2 -23677.137} C_VEL
LIN {X 0,Y 315.043,Z 370.158,A -85,B 0,C 180,E1 -23678.984,E2 -23678.984} C_VEL
LIN {X 0,Y 311.816,Z 367.97,A -85,B 0,C 180,E1 -23680.388,E2 -23680.388} C_VEL
LIN {X 0,Y 307.83,Z 365.284,A -85,B 0,C 180,E1 -23681.857,E2 -23681.857} C_VEL
LIN {X 0,Y 302.565,Z 361.993,A -85,B 0,C 180,E1 -23683.431,E2 -23683.431} C_VEL
LIN {X 0,Y 296.431,Z 357.74,A -85,B 0,C 180,E1 -23685.117,E2 -23685.117} C_VEL
LIN {X 0,Y 289.818,Z 353.141,A -85,B 0,C 180,E1 -23686.697,E2 -23686.697} C_VEL
LIN {X 0,Y 278.837,Z 345.675,A -85,B 0,C 180,E1 -23689.127,E2 -23689.127} C_VEL
LIN {X 0,Y 265.341,Z 336.573,A -85,B 0,C 180,E1 -23692.025,E2 -23692.025} C_VEL
LIN {X 0,Y 252.116,Z 326.576,A -85,B 0,C 180,E1 -23695.046,E2 -23695.046} C_VEL
LIN {X 0,Y 241.109,Z 316.705,A -85,B 0,C 180,E1 -23697.799,E2 -23697.799} C_VEL
LIN {X 0,Y 230.684,Z 305.429,A -85,B 0,C 180,E1 -23700.624,E2 -23700.624} C_VEL
LIN {X 0,Y 221.647,Z 294.174,A -85,B 0,C 180,E1 -23703.147,E2 -23703.147} C_VEL
LIN {X 0,Y 214.577,Z 284.271,A -85,B 0,C 180,E1 -23705.137,E2 -23705.137} C_VEL
LIN {X 0,Y 205.977,Z 270.615,A -85,B 0,C 180,E1 -23707.513,E2 -23707.513} C_VEL
LIN {X 0,Y 198.395,Z 255.928,A -85,B 0,C 180,E1 -23709.903,E2 -23709.903} C_VEL
LIN {X 0,Y 191.449,Z 240.113,A -85,B 0,C 180,E1 -23712.461,E2 -23712.461} C_VEL
LIN {X 0,Y 185.612,Z 228.344,A -85,B 0,C 180,E1 -23714.771,E2 -23714.771} C_VEL
LIN {X 0,Y 178.865,Z 216.851,A -85,B 0,C 180,E1 -23717.641,E2 -23717.641} C_VEL
LIN {X 0,Y 173.339,Z 208.611,A -85,B 0,C 180,E1 -23720.221,E2 -23720.221} C_VEL
LIN {X 0,Y 170.546,Z 204.641,A -85,B 0,C 180,E1 -23721.634,E2 -23721.634} C_VEL
LIN {X 0,Y 168.076,Z 201.16,A -85,B 0,C 180,E1 -23722.96,E2 -23722.96} C_VEL
LIN {X 0,Y 165.415,Z 197.403,A -85,B 0,C 180,E1 -23724.484,E2 -23724.484} C_VEL
LIN {X 0,Y 162.348,Z 193.895,A -85,B 0,C 180,E1 -23726.315,E2 -23726.315} C_VEL
LIN {X 0,Y 161.124,Z 191.81,A -85,B 0,C 180,E1 -23727.147,E2 -23727.147} C_VEL
LIN {X 0,Y 158.713,Z 189.779,A -85,B 0,C 180,E1 -23728.705,E2 -23728.705} C_VEL
LIN {X 0,Y 157.448,Z 187.137,A -85,B 0,C 180,E1 -23729.858,E2 -23729.858} C_VEL
LIN {X 0,Y 157.281,Z 186.434,A -85,B 0,C 180,E1 -23730.928,E2 -23730.928} C_VEL
LIN {X 0,Y 157.319,Z 186.35,A -85,B 0,C 180,E1 -23733.467,E2 -23733.467} C_VEL
LIN {X 0,Y 157.391,Z 186.335,A -85,B 0,C 180,E1 -23739.669,E2 -23739.669} C_VEL
LIN {X 0,Y 157.476,Z 186.357,A -85,B 0,C 180,E1 -23744.47,E2 -23744.47} C_VEL
LIN {X 0,Y 157.725,Z 186.283,A -85,B 0,C 180,E1 -23749.735,E2 -23749.735} C_VEL
LIN {X 0,Y 157.784,Z 186.29,A -85,B 0,C 180,E1 -23752.322,E2 -23752.322} C_VEL
LIN {X 0,Y 158.255,Z 186.214,A -85,B 0,C 180,E1 -23760.001,E2 -23760.001} C_VEL
LIN {X 0,Y 157.767,Z 186.287,A -85,B 0,C 180,E1 -23767.681,E2 -23767.681} C_VEL
LIN {X 0,Y 157.637,Z 186.299,A -85,B 0,C 180,E1 -23771.238,E2 -23771.238} C_VEL
LIN {X 0,Y 157.453,Z 186.349,A -85,B 0,C 180,E1 -23775.536,E2 -23775.536} C_VEL
LIN {X 0,Y 157.37,Z 186.344,A -85,B 0,C 180,E1 -23780.934,E2 -23780.934} C_VEL
LIN {X 0,Y 157.311,Z 186.347,A -85,B 0,C 180,E1 -23786.683,E2 -23786.683} C_VEL
LIN {X 0,Y 157.338,Z 186.67,A -85,B 0,C 180,E1 -23789.339,E2 -23789.339} C_VEL
LIN {X 0,Y 157.684,Z 187.891,A -85,B 0,C 180,E1 -23790.095,E2 -23790.095} C_VEL
LIN {X 0,Y 159.437,Z 190.578,A -85,B 0,C 180,E1 -23791.411,E2 -23791.411} C_VEL
LIN {X 0,Y 161.462,Z 192.14,A -85,B 0,C 180,E1 -23792.686,E2 -23792.686} C_VEL
LIN {X 0,Y 163.323,Z 195.264,A -85,B 0,C 180,E1 -23793.923,E2 -23793.923} C_VEL
LIN {X 0,Y 165.354,Z 197.322,A -85,B 0,C 180,E1 -23795.101,E2 -23795.101} C_VEL
LIN {X 0,Y 167.965,Z 201.07,A -85,B 0,C 180,E1 -23796.603,E2 -23796.603} C_VEL
LIN {X 0,Y 172.402,Z 208.345,A -85,B 0,C 180,E1 -23799.004,E2 -23799.004} C_VEL
LIN {X 0,Y 176.657,Z 215.861,A -85,B 0,C 180,E1 -23801.122,E2 -23801.122} C_VEL
LIN {X 0,Y 182.463,Z 227.449,A -85,B 0,C 180,E1 -23803.803,E2 -23803.803} C_VEL
LIN {X 0,Y 188.141,Z 241.145,A -85,B 0,C 180,E1 -23806.277,E2 -23806.277} C_VEL
LIN {X 0,Y 189.721,Z 245.736,A -85,B 0,C 180,E1 -23806.961,E2 -23806.961} C_VEL
LIN {X 0,Y 190.636,Z 252.792,A -85,B 0,C 180,E1 -23807.569,E2 -23807.569} C_VEL
LIN {X 0,Y 188.211,Z 291.894,A -85,B 0,C 180,E1 -23808.946,E2 -23808.946} C_VEL
LIN {X 0,Y 186.858,Z 303.06,A -85,B 0,C 180,E1 -23809.58,E2 -23809.58} C_VEL
LIN {X 0,Y 184.385,Z 316.415,A -85,B 0,C 180,E1 -23810.679,E2 -23810.679} C_VEL
LIN {X 0,Y 181.499,Z 327.96,A -85,B 0,C 180,E1 -23812.069,E2 -23812.069} C_VEL
LIN {X 0,Y 178.79,Z 337.232,A -85,B 0,C 180,E1 -23813.52,E2 -23813.52} C_VEL
LIN {X 0,Y 175.718,Z 346.171,A -85,B 0,C 180,E1 -23815.254,E2 -23815.254} C_VEL
LIN {X 0,Y 172.434,Z 354.694,A -85,B 0,C 180,E1 -23817.314,E2 -23817.314} C_VEL
LIN {X 0,Y 169.465,Z 361.91,A -85,B 0,C 180,E1 -23819.468,E2 -23819.468} C_VEL
LIN {X 0,Y 166.758,Z 368.109,A -85,B 0,C 180,E1 -23821.698,E2 -23821.698} C_VEL
LIN {X 0,Y 163.882,Z 374.649,A -85,B 0,C 180,E1 -23824.606,E2 -23824.606} C_VEL
LIN {X 0,Y 161.716,Z 379.149,A -85,B 0,C 180,E1 -23826.975,E2 -23826.975} C_VEL
LIN {X 0,Y 159.063,Z 384.641,A -85,B 0,C 180,E1 -23830.648,E2 -23830.648} C_VEL
LIN {X 0,Y 156.988,Z 388.967,A -85,B 0,C 180,E1 -23834.419,E2 -23834.419} C_VEL
LIN {X 0,Y 156.067,Z 391.339,A -85,B 0,C 180,E1 -23836.988,E2 -23836.988} C_VEL
LIN {X 0,Y 155.399,Z 393.144,A -85,B 0,C 180,E1 -23839.578,E2 -23839.578} C_VEL
LIN {X 0,Y 154.754,Z 395.603,A -85,B 0,C 180,E1 -23844.789,E2 -23844.789} C_VEL
LIN {X 0,Y 154.715,Z 396.318,A -85,B 0,C 180,E1 -23847.983,E2 -23847.983} C_VEL
LIN {X 0,Y 154.687,Z 396.348,A -85,B 0,C 180,E1 -23851.695,E2 -23851.695} C_VEL
LIN {X 0,Y 154.694,Z 395.601,A -85,B 0,C 180,E1 -23855.213,E2 -23855.213} C_VEL
LIN {X 0,Y 155.353,Z 393.143,A -85,B 0,C 180,E1 -23860.425,E2 -23860.425} C_VEL
LIN {X 0,Y 156.505,Z 390.187,A -85,B 0,C 180,E1 -23864.299,E2 -23864.299} C_VEL
LIN {X 0,Y 158.285,Z 386.194,A -85,B 0,C 180,E1 -23868.108,E2 -23868.108} C_VEL
LIN {X 0,Y 160.771,Z 381.065,A -85,B 0,C 180,E1 -23871.812,E2 -23871.812} C_VEL
LIN {X 0,Y 163.347,Z 375.805,A -85,B 0,C 180,E1 -23874.802,E2 -23874.802} C_VEL
LIN {X 0,Y 166.149,Z 369.486,A -85,B 0,C 180,E1 -23877.729,E2 -23877.729} C_VEL
LIN {X 0,Y 166.623,Z 368.424,A -85,B 0,C 180,E1 -23878.171,E2 -23878.171} C_VEL
LIN {X 0,Y 167.683,Z 364.736,A -85,B 0,C 180,E1 -23879.712,E2 -23879.712} C_VEL
LIN {X 0,Y 167.936,Z 358.33,A -85,B 0,C 180,E1 -23882.302,E2 -23882.302} C_VEL
LIN {X 0,Y 168.367,Z 351.444,A -85,B 0,C 180,E1 -23884.723,E2 -23884.723} C_VEL
LIN {X 0,Y 169.572,Z 346.855,A -85,B 0,C 180,E1 -23885.916,E2 -23885.916} C_VEL
LIN {X 0,Y 172.6,Z 338.389,A -85,B 0,C 180,E1 -23887.645,E2 -23887.645} C_VEL
LIN {X 0,Y 175.459,Z 329.399,A -85,B 0,C 180,E1 -23889.114,E2 -23889.114} C_VEL
LIN {X 0,Y 178.188,Z 319.264,A -85,B 0,C 180,E1 -23890.415,E2 -23890.415} C_VEL
LIN {X 0,Y 180.793,Z 307.213,A -85,B 0,C 180,E1 -23891.568,E2 -23891.568} C_VEL
LIN {X 0,Y 182.657,Z 293.895,A -85,B 0,C 180,E1 -23892.428,E2 -23892.428} C_VEL
LIN {X 0,Y 184.177,Z 273.194,A -85,B 0,C 180,E1 -23893.208,E2 -23893.208} C_VEL
LIN {X 0,Y 185.333,Z 253.46,A -85,B 0,C 180,E1 -23893.903,E2 -23893.903} C_VEL
LIN {X 0,Y 184.447,Z 247.467,A -85,B 0,C 180,E1 -23894.485,E2 -23894.485} C_VEL
LIN {X 0,Y 179.172,Z 233.936,A -85,B 0,C 180,E1 -23896.925,E2 -23896.925} C_VEL
LIN {X 0,Y 173.855,Z 222.782,A -85,B 0,C 180,E1 -23899.508,E2 -23899.508} C_VEL
LIN {X 0,Y 169.493,Z 214.598,A -85,B 0,C 180,E1 -23901.798,E2 -23901.798} C_VEL
LIN {X 0,Y 166.823,Z 210.024,A -85,B 0,C 180,E1 -23903.291,E2 -23903.291} C_VEL
LIN {X 0,Y 164.591,Z 206.365,A -85,B 0,C 180,E1 -23904.607,E2 -23904.607} C_VEL
LIN {X 0,Y 161.843,Z 202.546,A -85,B 0,C 180,E1 -23906.286,E2 -23906.286} C_VEL
LIN {X 0,Y 159.202,Z 199.126,A -85,B 0,C 180,E1 -23908.01,E2 -23908.01} C_VEL
LIN {X 0,Y 158.442,Z 198,A -85,B 0,C 180,E1 -23908.545,E2 -23908.545} C_VEL
LIN {X 0,Y 155.968,Z 195.419,A -85,B 0,C 180,E1 -23910.285,E2 -23910.285} C_VEL
LIN {X 0,Y 154.515,Z 192.925,A -85,B 0,C 180,E1 -23911.471,E2 -23911.471} C_VEL
LIN {X 0,Y 151.885,Z 190.885,A -85,B 0,C 180,E1 -23913.547,E2 -23913.547} C_VEL
LIN {X 0,Y 150.49,Z 188.476,A -85,B 0,C 180,E1 -23914.946,E2 -23914.946} C_VEL
LIN {X 0,Y 150.275,Z 187.492,A -85,B 0,C 180,E1 -23915.843,E2 -23915.843} C_VEL
LIN {X 0,Y 150.341,Z 187.205,A -85,B 0,C 180,E1 -23920.898,E2 -23920.898} C_VEL
LIN {X 0,Y 150.436,Z 187.23,A -85,B 0,C 180,E1 -23926.49,E2 -23926.49} C_VEL
LIN {X 0,Y 150.611,Z 187.169,A -85,B 0,C 180,E1 -23929.241,E2 -23929.241} C_VEL
LIN {X 0,Y 150.704,Z 187.161,A -85,B 0,C 180,E1 -23931.956,E2 -23931.956} C_VEL
LIN {X 0,Y 151.216,Z 187.09,A -85,B 0,C 180,E1 -23939.999,E2 -23939.999} C_VEL
LIN {X 0,Y 150.723,Z 187.163,A -85,B 0,C 180,E1 -23948.04,E2 -23948.04} C_VEL
LIN {X 0,Y 150.61,Z 187.175,A -85,B 0,C 180,E1 -23951.499,E2 -23951.499} C_VEL
LIN {X 0,Y 150.38,Z 187.225,A -85,B 0,C 180,E1 -23956.283,E2 -23956.283} C_VEL
LIN {X 0,Y 150.349,Z 187.215,A -85,B 0,C 180,E1 -23960.791,E2 -23960.791} C_VEL
LIN {X 0,Y 150.261,Z 187.493,A -85,B 0,C 180,E1 -23964.616,E2 -23964.616} C_VEL
LIN {X 0,Y 150.544,Z 188.595,A -85,B 0,C 180,E1 -23965.505,E2 -23965.505} C_VEL
LIN {X 0,Y 152.17,Z 191.253,A -85,B 0,C 180,E1 -23967.084,E2 -23967.084} C_VEL
LIN {X 0,Y 154.788,Z 193.216,A -85,B 0,C 180,E1 -23969.121,E2 -23969.121} C_VEL
LIN {X 0,Y 156.751,Z 196.485,A -85,B 0,C 180,E1 -23970.683,E2 -23970.683} C_VEL
LIN {X 0,Y 158.909,Z 198.503,A -85,B 0,C 180,E1 -23972.149,E2 -23972.149} C_VEL
LIN {X 0,Y 161.388,Z 202.115,A -85,B 0,C 180,E1 -23973.818,E2 -23973.818} C_VEL
LIN {X 0,Y 162.748,Z 203.677,A -85,B 0,C 180,E1 -23974.651,E2 -23974.651} C_VEL
LIN {X 0,Y 166.629,Z 209.198,A -85,B 0,C 180,E1 -23976.942,E2 -23976.942} C_VEL
LIN {X 0,Y 169.445,Z 213.265,A -85,B 0,C 180,E1 -23978.472,E2 -23978.472} C_VEL
LIN {X 0,Y 175.862,Z 223.093,A -85,B 0,C 180,E1 -23981.646,E2 -23981.646} C_VEL
LIN {X 0,Y 182.911,Z 235.738,A -85,B 0,C 180,E1 -23984.784,E2 -23984.784} C_VEL
LIN {X 0,Y 189.069,Z 249.077,A -85,B 0,C 180,E1 -23987.327,E2 -23987.327} C_VEL
LIN {X 0,Y 197.414,Z 267.895,A -85,B 0,C 180,E1 -23990.414,E2 -23990.414} C_VEL
LIN {X 0,Y 205.386,Z 282.038,A -85,B 0,C 180,E1 -23992.911,E2 -23992.911} C_VEL
LIN {X 0,Y 211.649,Z 291.914,A -85,B 0,C 180,E1 -23994.853,E2 -23994.853} C_VEL
LIN {X 0,Y 219.329,Z 302.582,A -85,B 0,C 180,E1 -23997.258,E2 -23997.258} C_VEL
LIN {X 0,Y 227.668,Z 312.732,A -85,B 0,C 180,E1 -23999.806,E2 -23999.806} C_VEL
LIN {X 0,Y 237.415,Z 322.956,A -85,B 0,C 180,E1 -24002.629,E2 -24002.629} C_VEL
LIN {X 0,Y 247.526,Z 331.769,A -85,B 0,C 180,E1 -24005.307,E2 -24005.307} C_VEL
LIN {X 0,Y 260.657,Z 341.432,A -85,B 0,C 180,E1 -24008.465,E2 -24008.465} C_VEL
LIN {X 0,Y 274.191,Z 350.188,A -85,B 0,C 180,E1 -24011.506,E2 -24011.506} C_VEL
LIN {X 0,Y 286.596,Z 358.156,A -85,B 0,C 180,E1 -24014.351,E2 -24014.351} C_VEL
LIN {X 0,Y 293.532,Z 362.975,A -85,B 0,C 180,E1 -24016.147,E2 -24016.147} C_VEL
LIN {X 0,Y 299.382,Z 366.841,A -85,B 0,C 180,E1 -24017.803,E2 -24017.803} C_VEL
LIN {X 0,Y 304.112,Z 369.804,A -85,B 0,C 180,E1 -24019.346,E2 -24019.346} C_VEL
LIN {X 0,Y 307.632,Z 372.245,A -85,B 0,C 180,E1 -24020.798,E2 -24020.798} C_VEL
LIN {X 0,Y 311.691,Z 374.869,A -85,B 0,C 180,E1 -24022.792,E2 -24022.792} C_VEL
LIN {X 0,Y 315.287,Z 376.744,A -85,B 0,C 180,E1 -24024.885,E2 -24024.885} C_VEL
LIN {X 0,Y 317.044,Z 377.489,A -85,B 0,C 180,E1 -24026.187,E2 -24026.187} C_VEL
LIN {X 0,Y 318.352,Z 377.992,A -85,B 0,C 180,E1 -24027.469,E2 -24027.469} C_VEL
LIN {X 0,Y 319.068,Z 378.311,A -85,B 0,C 180,E1 -24028.738,E2 -24028.738} C_VEL
LIN {X 0,Y 319.441,Z 378.367,A -85,B 0,C 180,E1 -24030,E2 -24030} C_VEL
LIN {X 0,Y 319.077,Z 378.305,A -85,B 0,C 180,E1 -24031.262,E2 -24031.262} C_VEL
LIN {X 0,Y 318.356,Z 377.988,A -85,B 0,C 180,E1 -24032.531,E2 -24032.531} C_VEL
LIN {X 0,Y 316.981,Z 377.457,A -85,B 0,C 180,E1 -24033.878,E2 -24033.878} C_VEL
LIN {X 0,Y 315.279,Z 376.748,A -85,B 0,C 180,E1 -24035.116,E2 -24035.116} C_VEL
LIN {X 0,Y 311.706,Z 374.809,A -85,B 0,C 180,E1 -24037.231,E2 -24037.231} C_VEL
LIN {X 0,Y 307.615,Z 372.232,A -85,B 0,C 180,E1 -24039.203,E2 -24039.203} C_VEL
LIN {X 0,Y 304.087,Z 369.798,A -85,B 0,C 180,E1 -24040.655,E2 -24040.655} C_VEL
LIN {X 0,Y 298.202,Z 366.129,A -85,B 0,C 180,E1 -24042.544,E2 -24042.544} C_VEL
LIN {X 0,Y 290.559,Z 360.891,A -85,B 0,C 180,E1 -24044.648,E2 -24044.648} C_VEL
LIN {X 0,Y 282.365,Z 355.532,A -85,B 0,C 180,E1 -24046.617,E2 -24046.617} C_VEL
LIN {X 0,Y 271.456,Z 348.509,A -85,B 0,C 180,E1 -24049.097,E2 -24049.097} C_VEL
LIN {X 0,Y 257.983,Z 339.594,A -85,B 0,C 180,E1 -24052.148,E2 -24052.148} C_VEL
LIN {X 0,Y 244.956,Z 329.676,A -85,B 0,C 180,E1 -24055.347,E2 -24055.347} C_VEL
LIN {X 0,Y 234.943,Z 320.535,A -85,B 0,C 180,E1 -24058.063,E2 -24058.063} C_VEL
LIN {X 0,Y 225.213,Z 309.807,A -85,B 0,C 180,E1 -24060.948,E2 -24060.948} C_VEL
LIN {X 0,Y 217.118,Z 299.532,A -85,B 0,C 180,E1 -24063.456,E2 -24063.456} C_VEL
LIN {X 0,Y 209.322,Z 288.253,A -85,B 0,C 180,E1 -24065.906,E2 -24065.906} C_VEL
LIN {X 0,Y 201.528,Z 275.444,A -85,B 0,C 180,E1 -24068.281,E2 -24068.281} C_VEL
LIN {X 0,Y 194.431,Z 261.65,A -85,B 0,C 180,E1 -24070.619,E2 -24070.619} C_VEL
LIN {X 0,Y 186.731,Z 243.834,A -85,B 0,C 180,E1 -24073.615,E2 -24073.615} C_VEL
LIN {X 0,Y 181.365,Z 232.831,A -85,B 0,C 180,E1 -24075.876,E2 -24075.876} C_VEL
LIN {X 0,Y 175.072,Z 221.829,A -85,B 0,C 180,E1 -24078.725,E2 -24078.725} C_VEL
LIN {X 0,Y 168.113,Z 211.174,A -85,B 0,C 180,E1 -24082.25,E2 -24082.25} C_VEL
LIN {X 0,Y 164.804,Z 206.63,A -85,B 0,C 180,E1 -24084.104,E2 -24084.104} C_VEL
LIN {X 0,Y 161.942,Z 202.668,A -85,B 0,C 180,E1 -24085.845,E2 -24085.845} C_VEL
LIN {X 0,Y 159.304,Z 199.273,A -85,B 0,C 180,E1 -24087.56,E2 -24087.56} C_VEL
LIN {X 0,Y 158.408,Z 197.975,A -85,B 0,C 180,E1 -24088.187,E2 -24088.187} C_VEL
LIN {X 0,Y 155.936,Z 195.412,A -85,B 0,C 180,E1 -24089.926,E2 -24089.926} C_VEL
LIN {X 0,Y 154.501,Z 192.929,A -85,B 0,C 180,E1 -24091.1,E2 -24091.1} C_VEL
LIN {X 0,Y 151.871,Z 190.915,A -85,B 0,C 180,E1 -24093.174,E2 -24093.174} C_VEL
LIN {X 0,Y 150.368,Z 187.987,A -85,B 0,C 180,E1 -24094.861,E2 -24094.861} C_VEL
LIN {X 0,Y 150.264,Z 187.3,A -85,B 0,C 180,E1 -24096.211,E2 -24096.211} C_VEL
LIN {X 0,Y 150.365,Z 187.205,A -85,B 0,C 180,E1 -24100.904,E2 -24100.904} C_VEL
LIN {X 0,Y 150.458,Z 187.224,A -85,B 0,C 180,E1 -24106.495,E2 -24106.495} C_VEL
LIN {X 0,Y 150.651,Z 187.165,A -85,B 0,C 180,E1 -24109.247,E2 -24109.247} C_VEL
LIN {X 0,Y 150.723,Z 187.163,A -85,B 0,C 180,E1 -24111.96,E2 -24111.96} C_VEL
LIN {X 0,Y 151.216,Z 187.09,A -85,B 0,C 180,E1 -24120.001,E2 -24120.001} C_VEL
LIN {X 0,Y 150.704,Z 187.161,A -85,B 0,C 180,E1 -24128.044,E2 -24128.044} C_VEL
LIN {X 0,Y 150.577,Z 187.179,A -85,B 0,C 180,E1 -24131.438,E2 -24131.438} C_VEL
LIN {X 0,Y 150.361,Z 187.218,A -85,B 0,C 180,E1 -24136.288,E2 -24136.288} C_VEL
LIN {X 0,Y 150.351,Z 187.215,A -85,B 0,C 180,E1 -24140.793,E2 -24140.793} C_VEL
LIN {X 0,Y 150.286,Z 187.521,A -85,B 0,C 180,E1 -24144.247,E2 -24144.247} C_VEL
LIN {X 0,Y 150.579,Z 188.703,A -85,B 0,C 180,E1 -24145.17,E2 -24145.17} C_VEL
LIN {X 0,Y 152.007,Z 191.06,A -85,B 0,C 180,E1 -24146.562,E2 -24146.562} C_VEL
LIN {X 0,Y 154.794,Z 193.285,A -85,B 0,C 180,E1 -24148.751,E2 -24148.751} C_VEL
LIN {X 0,Y 156.856,Z 196.597,A -85,B 0,C 180,E1 -24150.379,E2 -24150.379} C_VEL
LIN {X 0,Y 158.926,Z 198.604,A -85,B 0,C 180,E1 -24151.788,E2 -24151.788} C_VEL
LIN {X 0,Y 161.508,Z 202.236,A -85,B 0,C 180,E1 -24153.512,E2 -24153.512} C_VEL
LIN {X 0,Y 162.82,Z 203.833,A -85,B 0,C 180,E1 -24154.32,E2 -24154.32} C_VEL
LIN {X 0,Y 165.763,Z 208.148,A -85,B 0,C 180,E1 -24156.084,E2 -24156.084} C_VEL
LIN {X 0,Y 169.117,Z 213.913,A -85,B 0,C 180,E1 -24157.994,E2 -24157.994} C_VEL
LIN {X 0,Y 173.732,Z 222.567,A -85,B 0,C 180,E1 -24160.431,E2 -24160.431} C_VEL
LIN {X 0,Y 178.658,Z 232.755,A -85,B 0,C 180,E1 -24162.832,E2 -24162.832} C_VEL
LIN {X 0,Y 183.922,Z 245.981,A -85,B 0,C 180,E1 -24165.275,E2 -24165.275} C_VEL
LIN {X 0,Y 184.806,Z 248.968,A -85,B 0,C 180,E1 -24165.703,E2 -24165.703} C_VEL
LIN {X 0,Y 185.352,Z 254.461,A -85,B 0,C 180,E1 -24166.155,E2 -24166.155} C_VEL
LIN {X 0,Y 182.929,Z 291.732,A -85,B 0,C 180,E1 -24167.491,E2 -24167.491} C_VEL
LIN {X 0,Y 181.523,Z 302.845,A -85,B 0,C 180,E1 -24168.128,E2 -24168.128} C_VEL
LIN {X 0,Y 178.958,Z 316.224,A -85,B 0,C 180,E1 -24169.241,E2 -24169.241} C_VEL
LIN {X 0,Y 175.954,Z 327.768,A -85,B 0,C 180,E1 -24170.649,E2 -24170.649} C_VEL
LIN {X 0,Y 173.125,Z 337.04,A -85,B 0,C 180,E1 -24172.121,E2 -24172.121} C_VEL
LIN {X 0,Y 169.931,Z 345.98,A -85,B 0,C 180,E1 -24173.889,E2 -24173.889} C_VEL
LIN {X 0,Y 166.5,Z 354.502,A -85,B 0,C 180,E1 -24175.994,E2 -24175.994} C_VEL
LIN {X 0,Y 163.362,Z 361.717,A -85,B 0,C 180,E1 -24178.197,E2 -24178.197} C_VEL
LIN {X 0,Y 160.51,Z 367.917,A -85,B 0,C 180,E1 -24180.49,E2 -24180.49} C_VEL
LIN {X 0,Y 157.425,Z 374.455,A -85,B 0,C 180,E1 -24183.485,E2 -24183.485} C_VEL
LIN {X 0,Y 155.198,Z 378.957,A -85,B 0,C 180,E1 -24185.949,E2 -24185.949} C_VEL
LIN {X 0,Y 152.354,Z 384.448,A -85,B 0,C 180,E1 -24189.759,E2 -24189.759} C_VEL
LIN {X 0,Y 150.122,Z 388.774,A -85,B 0,C 180,E1 -24193.687,E2 -24193.687} C_VEL
LIN {X 0,Y 149.122,Z 391.147,A -85,B 0,C 180,E1 -24196.37,E2 -24196.37} C_VEL
LIN {X 0,Y 148.385,Z 392.951,A -85,B 0,C 180,E1 -24199.079,E2 -24199.079} C_VEL
LIN {X 0,Y 147.686,Z 395.411,A -85,B 0,C 180,E1 -24204.539,E2 -24204.539} C_VEL
LIN {X 0,Y 147.628,Z 396.162,A -85,B 0,C 180,E1 -24208.73,E2 -24208.73} C_VEL
LIN {X 0,Y 147.571,Z 396.005,A -85,B 0,C 180,E1 -24212.73,E2 -24212.73} C_VEL
LIN {X 0,Y 147.621,Z 395.409,A -85,B 0,C 180,E1 -24215.464,E2 -24215.464} C_VEL
LIN {X 0,Y 148.349,Z 392.95,A -85,B 0,C 180,E1 -24220.923,E2 -24220.923} C_VEL
LIN {X 0,Y 149.608,Z 389.994,A -85,B 0,C 180,E1 -24224.973,E2 -24224.973} C_VEL
LIN {X 0,Y 151.541,Z 386.002,A -85,B 0,C 180,E1 -24228.943,E2 -24228.943} C_VEL
LIN {X 0,Y 154.159,Z 380.872,A -85,B 0,C 180,E1 -24232.799,E2 -24232.799} C_VEL
LIN {X 0,Y 156.903,Z 375.612,A -85,B 0,C 180,E1 -24235.895,E2 -24235.895} C_VEL
LIN {X 0,Y 159.082,Z 371.025,A -85,B 0,C 180,E1 -24238.168,E2 -24238.168} C_VEL
LIN {X 0,Y 161.9,Z 364.97,A -85,B 0,C 180,E1 -24240.667,E2 -24240.667} C_VEL
LIN {X 0,Y 165.719,Z 356.421,A -85,B 0,C 180,E1 -24243.457,E2 -24243.457} C_VEL
LIN {X 0,Y 169.041,Z 348.247,A -85,B 0,C 180,E1 -24245.595,E2 -24245.595} C_VEL
LIN {X 0,Y 169.572,Z 346.855,A -85,B 0,C 180,E1 -24245.916,E2 -24245.916} C_VEL
LIN {X 0,Y 170.799,Z 342.221,A -85,B 0,C 180,E1 -24247.056,E2 -24247.056} C_VEL
LIN {X 0,Y 171.22,Z 334.349,A -85,B 0,C 180,E1 -24249.087,E2 -24249.087} C_VEL
LIN {X 0,Y 171.488,Z 326.172,A -85,B 0,C 180,E1 -24250.924,E2 -24250.924} C_VEL
LIN {X 0,Y 172.415,Z 320.787,A -85,B 0,C 180,E1 -24251.734,E2 -24251.734} C_VEL
LIN {X 0,Y 174.719,Z 311.009,A -85,B 0,C 180,E1 -24252.748,E2 -24252.748} C_VEL
LIN {X 0,Y 176.472,Z 301.375,A -85,B 0,C 180,E1 -24253.503,E2 -24253.503} C_VEL
LIN {X 0,Y 177.748,Z 291.01,A -85,B 0,C 180,E1 -24254.091,E2 -24254.091} C_VEL
LIN {X 0,Y 180.208,Z 254.723,A -85,B 0,C 180,E1 -24255.412,E2 -24255.412} C_VEL
LIN {X 0,Y 179.449,Z 249.998,A -85,B 0,C 180,E1 -24255.921,E2 -24255.921} C_VEL
LIN {X 0,Y 174.42,Z 236.996,A -85,B 0,C 180,E1 -24258.425,E2 -24258.425} C_VEL
LIN {X 0,Y 169.447,Z 226.321,A -85,B 0,C 180,E1 -24261.04,E2 -24261.04} C_VEL
LIN {X 0,Y 165.07,Z 217.901,A -85,B 0,C 180,E1 -24263.543,E2 -24263.543} C_VEL
LIN {X 0,Y 161.579,Z 212.056,A -85,B 0,C 180,E1 -24265.688,E2 -24265.688} C_VEL
LIN {X 0,Y 159.06,Z 208.463,A -85,B 0,C 180,E1 -24267.323,E2 -24267.323} C_VEL
LIN {X 0,Y 155.69,Z 203.983,A -85,B 0,C 180,E1 -24269.691,E2 -24269.691} C_VEL
LIN {X 0,Y 153.135,Z 200.832,A -85,B 0,C 180,E1 -24271.657,E2 -24271.657} C_VEL
LIN {X 0,Y 152.164,Z 199.284,A -85,B 0,C 180,E1 -24272.491,E2 -24272.491} C_VEL
LIN {X 0,Y 149.559,Z 196.925,A -85,B 0,C 180,E1 -24274.713,E2 -24274.713} C_VEL
LIN {X 0,Y 147.804,Z 193.947,A -85,B 0,C 180,E1 -24276.531,E2 -24276.531} C_VEL
LIN {X 0,Y 145.29,Z 192.207,A -85,B 0,C 180,E1 -24279.141,E2 -24279.141} C_VEL
LIN {X 0,Y 143.689,Z 189.727,A -85,B 0,C 180,E1 -24281.276,E2 -24281.276} C_VEL
LIN {X 0,Y 143.329,Z 188.492,A -85,B 0,C 180,E1 -24282.521,E2 -24282.521} C_VEL
LIN {X 0,Y 143.359,Z 188.124,A -85,B 0,C 180,E1 -24285.81,E2 -24285.81} C_VEL
LIN {X 0,Y 143.537,Z 188.053,A -85,B 0,C 180,E1 -24288.704,E2 -24288.704} C_VEL
LIN {X 0,Y 143.626,Z 188.039,A -85,B 0,C 180,E1 -24291.557,E2 -24291.557} C_VEL
LIN {X 0,Y 144.174,Z 187.966,A -85,B 0,C 180,E1 -24299.998,E2 -24299.998} C_VEL
LIN {X 0,Y 143.647,Z 188.04,A -85,B 0,C 180,E1 -24308.439,E2 -24308.439} C_VEL
LIN {X 0,Y 143.547,Z 188.056,A -85,B 0,C 180,E1 -24311.711,E2 -24311.711} C_VEL
LIN {X 0,Y 143.346,Z 188.375,A -85,B 0,C 180,E1 -24317.658,E2 -24317.658} C_VEL
LIN {X 0,Y 143.653,Z 189.472,A -85,B 0,C 180,E1 -24319.003,E2 -24319.003} C_VEL
LIN {X 0,Y 145.088,Z 191.998,A -85,B 0,C 180,E1 -24321.002,E2 -24321.002} C_VEL
LIN {X 0,Y 147.461,Z 193.793,A -85,B 0,C 180,E1 -24323.524,E2 -24323.524} C_VEL
LIN {X 0,Y 148.11,Z 194.289,A -85,B 0,C 180,E1 -24324.157,E2 -24324.157} C_VEL
LIN {X 0,Y 150.055,Z 197.551,A -85,B 0,C 180,E1 -24326.129,E2 -24326.129} C_VEL
LIN {X 0,Y 152.608,Z 199.833,A -85,B 0,C 180,E1 -24328.259,E2 -24328.259} C_VEL
LIN {X 0,Y 154.783,Z 203.117,A -85,B 0,C 180,E1 -24330.034,E2 -24330.034} C_VEL
LIN {X 0,Y 156.647,Z 205.146,A -85,B 0,C 180,E1 -24331.379,E2 -24331.379} C_VEL
LIN {X 0,Y 159.376,Z 208.793,A -85,B 0,C 180,E1 -24333.259,E2 -24333.259} C_VEL
LIN {X 0,Y 163.662,Z 215.011,A -85,B 0,C 180,E1 -24335.957,E2 -24335.957} C_VEL
LIN {X 0,Y 168.571,Z 222.369,A -85,B 0,C 180,E1 -24338.708,E2 -24338.708} C_VEL
LIN {X 0,Y 174.433,Z 232.152,A -85,B 0,C 180,E1 -24341.666,E2 -24341.666} C_VEL
LIN {X 0,Y 179.861,Z 242.629,A -85,B 0,C 180,E1 -24344.179,E2 -24344.179} C_VEL
LIN {X 0,Y 185.479,Z 255.434,A -85,B 0,C 180,E1 -24346.623,E2 -24346.623} C_VEL
LIN {X 0,Y 192.867,Z 272.361,A -85,B 0,C 180,E1 -24349.496,E2 -24349.496} C_VEL
LIN {X 0,Y 200.754,Z 286.728,A -85,B 0,C 180,E1 -24352.171,E2 -24352.171} C_VEL
LIN {X 0,Y 207.272,Z 297.358,A -85,B 0,C 180,E1 -24354.464,E2 -24354.464} C_VEL
LIN {X 0,Y 215.785,Z 309.328,A -85,B 0,C 180,E1 -24357.433,E2 -24357.433} C_VEL
LIN {X 0,Y 224.468,Z 319.71,A -85,B 0,C 180,E1 -24360.321,E2 -24360.321} C_VEL
LIN {X 0,Y 233.751,Z 329.16,A -85,B 0,C 180,E1 -24363.193,E2 -24363.193} C_VEL
LIN {X 0,Y 242.848,Z 336.803,A -85,B 0,C 180,E1 -24365.728,E2 -24365.728} C_VEL
LIN {X 0,Y 255.903,Z 346.079,A -85,B 0,C 180,E1 -24369.026,E2 -24369.026} C_VEL
LIN {X 0,Y 269.436,Z 354.437,A -85,B 0,C 180,E1 -24372.183,E2 -24372.183} C_VEL
LIN {X 0,Y 280.403,Z 361.092,A -85,B 0,C 180,E1 -24374.784,E2 -24374.784} C_VEL
LIN {X 0,Y 288.563,Z 366.422,A -85,B 0,C 180,E1 -24376.954,E2 -24376.954} C_VEL
LIN {X 0,Y 294.024,Z 369.895,A -85,B 0,C 180,E1 -24378.521,E2 -24378.521} C_VEL
LIN {X 0,Y 297.996,Z 372.426,A -85,B 0,C 180,E1 -24379.813,E2 -24379.813} C_VEL
LIN {X 0,Y 302.953,Z 375.856,A -85,B 0,C 180,E1 -24381.999,E2 -24381.999} C_VEL
LIN {X 0,Y 305.772,Z 377.537,A -85,B 0,C 180,E1 -24383.401,E2 -24383.401} C_VEL
LIN {X 0,Y 308.108,Z 378.755,A -85,B 0,C 180,E1 -24384.765,E2 -24384.765} C_VEL
LIN {X 0,Y 310.034,Z 379.661,A -85,B 0,C 180,E1 -24386.101,E2 -24386.101} C_VEL
LIN {X 0,Y 311.461,Z 380.219,A -85,B 0,C 180,E1 -24387.413,E2 -24387.413} C_VEL
LIN {X 0,Y 312.289,Z 380.549,A -85,B 0,C 180,E1 -24388.71,E2 -24388.71} C_VEL
LIN {X 0,Y 312.71,Z 380.615,A -85,B 0,C 180,E1 -24390,E2 -24390} C_VEL
LIN {X 0,Y 312.296,Z 380.549,A -85,B 0,C 180,E1 -24391.289,E2 -24391.289} C_VEL
LIN {X 0,Y 311.466,Z 380.222,A -85,B 0,C 180,E1 -24392.587,E2 -24392.587} C_VEL
LIN {X 0,Y 309.97,Z 379.628,A -85,B 0,C 180,E1 -24393.966,E2 -24393.966} C_VEL
LIN {X 0,Y 308.104,Z 378.775,A -85,B 0,C 180,E1 -24395.235,E2 -24395.235} C_VEL
LIN {X 0,Y 304.62,Z 376.823,A -85,B 0,C 180,E1 -24397.227,E2 -24397.227} C_VEL
LIN {X 0,Y 299.759,Z 373.646,A -85,B 0,C 180,E1 -24399.446,E2 -24399.446} C_VEL
LIN {X 0,Y 297.96,Z 372.43,A -85,B 0,C 180,E1 -24400.189,E2 -24400.189} C_VEL
LIN {X 0,Y 291.577,Z 368.392,A -85,B 0,C 180,E1 -24402.199,E2 -24402.199} C_VEL
LIN {X 0,Y 283.128,Z 362.851,A -85,B 0,C 180,E1 -24404.518,E2 -24404.518} C_VEL
LIN {X 0,Y 272.163,Z 356.147,A -85,B 0,C 180,E1 -24407.172,E2 -24407.172} C_VEL
LIN {X 0,Y 258.578,Z 347.79,A -85,B 0,C 180,E1 -24410.338,E2 -24410.338} C_VEL
LIN {X 0,Y 245.149,Z 338.57,A -85,B 0,C 180,E1 -24413.663,E2 -24413.663} C_VEL
LIN {X 0,Y 235.299,Z 330.559,A -85,B 0,C 180,E1 -24416.359,E2 -24416.359} C_VEL
LIN {X 0,Y 226.835,Z 322.306,A -85,B 0,C 180,E1 -24418.92,E2 -24418.92} C_VEL
LIN {X 0,Y 218.649,Z 312.879,A -85,B 0,C 180,E1 -24421.596,E2 -24421.596} C_VEL
LIN {X 0,Y 211.791,Z 303.863,A -85,B 0,C 180,E1 -24423.945,E2 -24423.945} C_VEL
LIN {X 0,Y 205.415,Z 294.448,A -85,B 0,C 180,E1 -24426.176,E2 -24426.176} C_VEL
LIN {X 0,Y 198.446,Z 282.721,A -85,B 0,C 180,E1 -24428.618,E2 -24428.618} C_VEL
LIN {X 0,Y 190.589,Z 267.567,A -85,B 0,C 180,E1 -24431.332,E2 -24431.332} C_VEL
LIN {X 0,Y 182.181,Z 247.788,A -85,B 0,C 180,E1 -24434.788,E2 -24434.788} C_VEL
LIN {X 0,Y 177.165,Z 237.238,A -85,B 0,C 180,E1 -24437.046,E2 -24437.046} C_VEL
LIN {X 0,Y 171.371,Z 226.906,A -85,B 0,C 180,E1 -24439.84,E2 -24439.84} C_VEL
LIN {X 0,Y 165.045,Z 216.906,A -85,B 0,C 180,E1 -24443.246,E2 -24443.246} C_VEL
LIN {X 0,Y 161.654,Z 212.097,A -85,B 0,C 180,E1 -24445.266,E2 -24445.266} C_VEL
LIN {X 0,Y 159.05,Z 208.476,A -85,B 0,C 180,E1 -24446.947,E2 -24446.947} C_VEL
LIN {X 0,Y 156.322,Z 204.591,A -85,B 0,C 180,E1 -24448.868,E2 -24448.868} C_VEL
LIN {X 0,Y 153.391,Z 201.293,A -85,B 0,C 180,E1 -24451.058,E2 -24451.058} C_VEL
LIN {X 0,Y 152.341,Z 199.446,A -85,B 0,C 180,E1 -24451.969,E2 -24451.969} C_VEL
LIN {X 0,Y 149.696,Z 197.084,A -85,B 0,C 180,E1 -24454.206,E2 -24454.206} C_VEL
LIN {X 0,Y 147.792,Z 193.96,A -85,B 0,C 180,E1 -24456.161,E2 -24456.161} C_VEL
LIN {X 0,Y 145.349,Z 192.281,A -85,B 0,C 180,E1 -24458.691,E2 -24458.691} C_VEL
LIN {X 0,Y 143.742,Z 189.774,A -85,B 0,C 180,E1 -24460.824,E2 -24460.824} C_VEL
LIN {X 0,Y 143.398,Z 188.672,A -85,B 0,C 180,E1 -24461.795,E2 -24461.795} C_VEL
LIN {X 0,Y 143.344,Z 188.124,A -85,B 0,C 180,E1 -24464.358,E2 -24464.358} C_VEL
LIN {X 0,Y 143.593,Z 188.046,A -85,B 0,C 180,E1 -24468.712,E2 -24468.712} C_VEL
LIN {X 0,Y 143.647,Z 188.04,A -85,B 0,C 180,E1 -24471.561,E2 -24471.561} C_VEL
LIN {X 0,Y 144.174,Z 187.966,A -85,B 0,C 180,E1 -24480.002,E2 -24480.002} C_VEL
LIN {X 0,Y 143.626,Z 188.039,A -85,B 0,C 180,E1 -24488.443,E2 -24488.443} C_VEL
LIN {X 0,Y 143.505,Z 188.061,A -85,B 0,C 180,E1 -24491.63,E2 -24491.63} C_VEL
LIN {X 0,Y 143.312,Z 188.395,A -85,B 0,C 180,E1 -24497.297,E2 -24497.297} C_VEL
LIN {X 0,Y 143.647,Z 189.562,A -85,B 0,C 180,E1 -24498.637,E2 -24498.637} C_VEL
LIN {X 0,Y 145.204,Z 192.099,A -85,B 0,C 180,E1 -24500.756,E2 -24500.756} C_VEL
LIN {X 0,Y 147.47,Z 193.807,A -85,B 0,C 180,E1 -24503.154,E2 -24503.154} C_VEL
LIN {X 0,Y 148.116,Z 194.331,A -85,B 0,C 180,E1 -24503.787,E2 -24503.787} C_VEL
LIN {X 0,Y 149.918,Z 197.376,A -85,B 0,C 180,E1 -24505.622,E2 -24505.622} C_VEL
LIN {X 0,Y 152.528,Z 199.717,A -85,B 0,C 180,E1 -24507.811,E2 -24507.811} C_VEL
LIN {X 0,Y 154.914,Z 203.243,A -85,B 0,C 180,E1 -24509.751,E2 -24509.751} C_VEL
LIN {X 0,Y 156.564,Z 205.069,A -85,B 0,C 180,E1 -24510.942,E2 -24510.942} C_VEL
LIN {X 0,Y 159.437,Z 208.861,A -85,B 0,C 180,E1 -24512.919,E2 -24512.919} C_VEL
LIN {X 0,Y 162.727,Z 213.864,A -85,B 0,C 180,E1 -24515.032,E2 -24515.032} C_VEL
LIN {X 0,Y 167.257,Z 221.96,A -85,B 0,C 180,E1 -24517.731,E2 -24517.731} C_VEL
LIN {X 0,Y 172.862,Z 233.43,A -85,B 0,C 180,E1 -24520.773,E2 -24520.773} C_VEL
LIN {X 0,Y 177.491,Z 244.664,A -85,B 0,C 180,E1 -24523.119,E2 -24523.119} C_VEL
LIN {X 0,Y 179.887,Z 251.669,A -85,B 0,C 180,E1 -24524.315,E2 -24524.315} C_VEL
LIN {X 0,Y 180.186,Z 256.131,A -85,B 0,C 180,E1 -24524.659,E2 -24524.659} C_VEL
LIN {X 0,Y 177.693,Z 292.212,A -85,B 0,C 180,E1 -24525.975,E2 -24525.975} C_VEL
LIN {X 0,Y 175.95,Z 304.932,A -85,B 0,C 180,E1 -24526.736,E2 -24526.736} C_VEL
LIN {X 0,Y 173.113,Z 318.066,A -85,B 0,C 180,E1 -24527.944,E2 -24527.944} C_VEL
LIN {X 0,Y 170.521,Z 327.576,A -85,B 0,C 180,E1 -24529.135,E2 -24529.135} C_VEL
LIN {X 0,Y 167.582,Z 336.849,A -85,B 0,C 180,E1 -24530.632,E2 -24530.632} C_VEL
LIN {X 0,Y 164.243,Z 345.788,A -85,B 0,C 180,E1 -24532.428,E2 -24532.428} C_VEL
LIN {X 0,Y 160.663,Z 354.311,A -85,B 0,C 180,E1 -24534.578,E2 -24534.578} C_VEL
LIN {X 0,Y 157.355,Z 361.525,A -85,B 0,C 180,E1 -24536.83,E2 -24536.83} C_VEL
LIN {X 0,Y 154.36,Z 367.725,A -85,B 0,C 180,E1 -24539.189,E2 -24539.189} C_VEL
LIN {X 0,Y 151.04,Z 374.262,A -85,B 0,C 180,E1 -24542.27,E2 -24542.27} C_VEL
LIN {X 0,Y 148.74,Z 378.765,A -85,B 0,C 180,E1 -24544.834,E2 -24544.834} C_VEL
LIN {X 0,Y 145.688,Z 384.256,A -85,B 0,C 180,E1 -24548.789,E2 -24548.789} C_VEL
LIN {X 0,Y 143.288,Z 388.582,A -85,B 0,C 180,E1 -24552.885,E2 -24552.885} C_VEL
LIN {X 0,Y 142.206,Z 390.954,A -85,B 0,C 180,E1 -24555.694,E2 -24555.694} C_VEL
LIN {X 0,Y 141.395,Z 392.759,A -85,B 0,C 180,E1 -24558.532,E2 -24558.532} C_VEL
LIN {X 0,Y 140.616,Z 395.219,A -85,B 0,C 180,E1 -24564.263,E2 -24564.263} C_VEL
LIN {X 0,Y 140.572,Z 395.972,A -85,B 0,C 180,E1 -24569.356,E2 -24569.356} C_VEL
LIN {X 0,Y 140.489,Z 395.813,A -85,B 0,C 180,E1 -24572.867,E2 -24572.867} C_VEL
LIN {X 0,Y 140.545,Z 395.217,A -85,B 0,C 180,E1 -24575.74,E2 -24575.74} C_VEL
LIN {X 0,Y 141.366,Z 392.758,A -85,B 0,C 180,E1 -24581.47,E2 -24581.47} C_VEL
LIN {X 0,Y 142.712,Z 389.801,A -85,B 0,C 180,E1 -24585.715,E2 -24585.715} C_VEL
LIN {X 0,Y 144.806,Z 385.81,A -85,B 0,C 180,E1 -24589.861,E2 -24589.861} C_VEL
LIN {X 0,Y 147.608,Z 380.679,A -85,B 0,C 180,E1 -24593.872,E2 -24593.872} C_VEL
LIN {X 0,Y 150.518,Z 375.42,A -85,B 0,C 180,E1 -24597.08,E2 -24597.08} C_VEL
LIN {X 0,Y 153.65,Z 369.1,A -85,B 0,C 180,E1 -24600.208,E2 -24600.208} C_VEL
LIN {X 0,Y 156.582,Z 363.151,A -85,B 0,C 180,E1 -24602.588,E2 -24602.588} C_VEL
LIN {X 0,Y 159.821,Z 356.229,A -85,B 0,C 180,E1 -24604.866,E2 -24604.866} C_VEL
LIN {X 0,Y 163.307,Z 348.055,A -85,B 0,C 180,E1 -24607.048,E2 -24607.048} C_VEL
LIN {X 0,Y 166.546,Z 339.548,A -85,B 0,C 180,E1 -24608.88,E2 -24608.88} C_VEL
LIN {X 0,Y 169.503,Z 330.838,A -85,B 0,C 180,E1 -24610.379,E2 -24610.379} C_VEL
LIN {X 0,Y 172.415,Z 320.787,A -85,B 0,C 180,E1 -24611.734,E2 -24611.734} C_VEL
LIN {X 0,Y 173.32,Z 315.431,A -85,B 0,C 180,E1 -24612.489,E2 -24612.489} C_VEL
LIN {X 0,Y 173.093,Z 306.491,A -85,B 0,C 180,E1 -24613.938,E2 -24613.938} C_VEL
LIN {X 0,Y 172.513,Z 297.387,A -85,B 0,C 180,E1 -24615.231,E2 -24615.231} C_VEL
LIN {X 0,Y 172.634,Z 291.643,A -85,B 0,C 180,E1 -24615.694,E2 -24615.694} C_VEL
LIN {X 0,Y 175.172,Z 257.225,A -85,B 0,C 180,E1 -24616.95,E2 -24616.95} C_VEL
LIN {X 0,Y 174.97,Z 253.72,A -85,B 0,C 180,E1 -24617.227,E2 -24617.227} C_VEL
LIN {X 0,Y 170.342,Z 241.343,A -85,B 0,C 180,E1 -24619.707,E2 -24619.707} C_VEL
LIN {X 0,Y 165.734,Z 231.08,A -85,B 0,C 180,E1 -24622.315,E2 -24622.315} C_VEL
LIN {X 0,Y 161.224,Z 222.144,A -85,B 0,C 180,E1 -24625.099,E2 -24625.099} C_VEL
LIN {X 0,Y 158.354,Z 217.29,A -85,B 0,C 180,E1 -24626.997,E2 -24626.997} C_VEL
LIN {X 0,Y 155.75,Z 213.631,A -85,B 0,C 180,E1 -24628.807,E2 -24628.807} C_VEL
LIN {X 0,Y 153.225,Z 210.09,A -85,B 0,C 180,E1 -24630.719,E2 -24630.719} C_VEL
LIN {X 0,Y 150.564,Z 206.564,A -85,B 0,C 180,E1 -24632.922,E2 -24632.922} C_VEL
LIN {X 0,Y 149.584,Z 205.408,A -85,B 0,C 180,E1 -24633.781,E2 -24633.781} C_VEL
LIN {X 0,Y 146.907,Z 202.315,A -85,B 0,C 180,E1 -24636.332,E2 -24636.332} C_VEL
LIN {X 0,Y 146.006,Z 200.654,A -85,B 0,C 180,E1 -24637.35,E2 -24637.35} C_VEL
LIN {X 0,Y 143.508,Z 198.622,A -85,B 0,C 180,E1 -24640.137,E2 -24640.137} C_VEL
LIN {X 0,Y 141.791,Z 195.715,A -85,B 0,C 180,E1 -24642.604,E2 -24642.604} C_VEL
LIN {X 0,Y 141.05,Z 194.909,A -85,B 0,C 180,E1 -24643.722,E2 -24643.722} C_VEL
LIN {X 0,Y 138.353,Z 192.93,A -85,B 0,C 180,E1 -24648.547,E2 -24648.547} C_VEL
LIN {X 0,Y 136.705,Z 189.689,A -85,B 0,C 180,E1 -24654.837,E2 -24654.837} C_VEL
LIN {X 0,Y 137.131,Z 188.971,A -85,B 0,C 180,E1 -24659.998,E2 -24659.998} C_VEL
LIN {X 0,Y 136.714,Z 189.575,A -85,B 0,C 180,E1 -24665.16,E2 -24665.16} C_VEL
LIN {X 0,Y 137.439,Z 191.554,A -85,B 0,C 180,E1 -24669.379,E2 -24669.379} C_VEL
LIN {X 0,Y 139.929,Z 194.342,A -85,B 0,C 180,E1 -24674.915,E2 -24674.915} C_VEL
LIN {X 0,Y 141.743,Z 195.491,A -85,B 0,C 180,E1 -24677.678,E2 -24677.678} C_VEL
LIN {X 0,Y 143.237,Z 198.311,A -85,B 0,C 180,E1 -24679.899,E2 -24679.899} C_VEL
LIN {X 0,Y 145.68,Z 200.472,A -85,B 0,C 180,E1 -24682.701,E2 -24682.701} C_VEL
LIN {X 0,Y 146.293,Z 201.082,A -85,B 0,C 180,E1 -24683.348,E2 -24683.348} C_VEL
LIN {X 0,Y 148.452,Z 204.39,A -85,B 0,C 180,E1 -24685.592,E2 -24685.592} C_VEL
LIN {X 0,Y 150.388,Z 206.229,A -85,B 0,C 180,E1 -24687.293,E2 -24687.293} C_VEL
LIN {X 0,Y 153.197,Z 210.088,A -85,B 0,C 180,E1 -24689.641,E2 -24689.641} C_VEL
LIN {X 0,Y 154.924,Z 212.508,A -85,B 0,C 180,E1 -24690.969,E2 -24690.969} C_VEL
LIN {X 0,Y 157.555,Z 216.071,A -85,B 0,C 180,E1 -24692.835,E2 -24692.835} C_VEL
LIN {X 0,Y 162.349,Z 223.125,A -85,B 0,C 180,E1 -24695.915,E2 -24695.915} C_VEL
LIN {X 0,Y 168.733,Z 233.635,A -85,B 0,C 180,E1 -24699.524,E2 -24699.524} C_VEL
LIN {X 0,Y 174.81,Z 245.224,A -85,B 0,C 180,E1 -24702.592,E2 -24702.592} C_VEL
LIN {X 0,Y 180.523,Z 258.379,A -85,B 0,C 180,E1 -24705.27,E2 -24705.27} C_VEL
LIN {X 0,Y 188.13,Z 276.325,A -85,B 0,C 180,E1 -24708.442,E2 -24708.442} C_VEL
LIN {X 0,Y 195.321,Z 290.135,A -85,B 0,C 180,E1 -24711.188,E2 -24711.188} C_VEL
LIN {X 0,Y 201.383,Z 300.664,A -85,B 0,C 180,E1 -24713.61,E2 -24713.61} C_VEL
LIN {X 0,Y 208.592,Z 311.392,A -85,B 0,C 180,E1 -24716.429,E2 -24716.429} C_VEL
LIN {X 0,Y 216.477,Z 321.4,A -85,B 0,C 180,E1 -24719.352,E2 -24719.352} C_VEL
LIN {X 0,Y 225.763,Z 331.282,A -85,B 0,C 180,E1 -24722.52,E2 -24722.52} C_VEL
LIN {X 0,Y 235.54,Z 339.783,A -85,B 0,C 180,E1 -24725.508,E2 -24725.508} C_VEL
LIN {X 0,Y 248.435,Z 348.906,A -85,B 0,C 180,E1 -24728.99,E2 -24728.99} C_VEL
LIN {X 0,Y 262.835,Z 357.433,A -85,B 0,C 180,E1 -24732.494,E2 -24732.494} C_VEL
LIN {X 0,Y 273.585,Z 363.574,A -85,B 0,C 180,E1 -24735.115,E2 -24735.115} C_VEL
LIN {X 0,Y 281.163,Z 368.092,A -85,B 0,C 180,E1 -24737.119,E2 -24737.119} C_VEL
LIN {X 0,Y 289.296,Z 372.999,A -85,B 0,C 180,E1 -24739.511,E2 -24739.511} C_VEL
LIN {X 0,Y 292.153,Z 374.774,A -85,B 0,C 180,E1 -24740.497,E2 -24740.497} C_VEL
LIN {X 0,Y 295.192,Z 376.871,A -85,B 0,C 180,E1 -24741.787,E2 -24741.787} C_VEL
LIN {X 0,Y 298.178,Z 378.829,A -85,B 0,C 180,E1 -24743.232,E2 -24743.232} C_VEL
LIN {X 0,Y 300.681,Z 380.185,A -85,B 0,C 180,E1 -24744.635,E2 -24744.635} C_VEL
LIN {X 0,Y 302.902,Z 381.261,A -85,B 0,C 180,E1 -24746.096,E2 -24746.096} C_VEL
LIN {X 0,Y 304.39,Z 381.911,A -85,B 0,C 180,E1 -24747.353,E2 -24747.353} C_VEL
LIN {X 0,Y 305.365,Z 382.3,A -85,B 0,C 180,E1 -24748.681,E2 -24748.681} C_VEL
LIN {X 0,Y 305.848,Z 382.384,A -85,B 0,C 180,E1 -24750,E2 -24750} C_VEL
LIN {X 0,Y 305.371,Z 382.301,A -85,B 0,C 180,E1 -24751.319,E2 -24751.319} C_VEL
LIN {X 0,Y 304.418,Z 381.914,A -85,B 0,C 180,E1 -24752.646,E2 -24752.646} C_VEL
LIN {X 0,Y 302.812,Z 381.219,A -85,B 0,C 180,E1 -24753.993,E2 -24753.993} C_VEL
LIN {X 0,Y 300.693,Z 380.212,A -85,B 0,C 180,E1 -24755.364,E2 -24755.364} C_VEL
LIN {X 0,Y 297.472,Z 378.371,A -85,B 0,C 180,E1 -24757.131,E2 -24757.131} C_VEL
LIN {X 0,Y 293.722,Z 375.877,A -85,B 0,C 180,E1 -24758.845,E2 -24758.845} C_VEL
LIN {X 0,Y 291.604,Z 374.405,A -85,B 0,C 180,E1 -24759.713,E2 -24759.713} C_VEL
LIN {X 0,Y 286.563,Z 371.364,A -85,B 0,C 180,E1 -24761.315,E2 -24761.315} C_VEL
LIN {X 0,Y 278.154,Z 366.254,A -85,B 0,C 180,E1 -24763.705,E2 -24763.705} C_VEL
LIN {X 0,Y 267.392,Z 360.085,A -85,B 0,C 180,E1 -24766.399,E2 -24766.399} C_VEL
LIN {X 0,Y 255.42,Z 353.171,A -85,B 0,C 180,E1 -24769.28,E2 -24769.28} C_VEL
LIN {X 0,Y 241.244,Z 344.057,A -85,B 0,C 180,E1 -24772.892,E2 -24772.892} C_VEL
LIN {X 0,Y 230.003,Z 335.176,A -85,B 0,C 180,E1 -24776.145,E2 -24776.145} C_VEL
LIN {X 0,Y 221.743,Z 327.217,A -85,B 0,C 180,E1 -24778.824,E2 -24778.824} C_VEL
LIN {X 0,Y 212.021,Z 315.887,A -85,B 0,C 180,E1 -24782.3,E2 -24782.3} C_VEL
LIN {X 0,Y 204.339,Z 305.208,A -85,B 0,C 180,E1 -24785.232,E2 -24785.232} C_VEL
LIN {X 0,Y 198.149,Z 295.127,A -85,B 0,C 180,E1 -24787.687,E2 -24787.687} C_VEL
LIN {X 0,Y 192.186,Z 284.263,A -85,B 0,C 180,E1 -24790.036,E2 -24790.036} C_VEL
LIN {X 0,Y 185.473,Z 270.528,A -85,B 0,C 180,E1 -24792.594,E2 -24792.594} C_VEL
LIN {X 0,Y 177.495,Z 251.152,A -85,B 0,C 180,E1 -24796.126,E2 -24796.126} C_VEL
LIN {X 0,Y 172.781,Z 241.142,A -85,B 0,C 180,E1 -24798.401,E2 -24798.401} C_VEL
LIN {X 0,Y 167.67,Z 231.786,A -85,B 0,C 180,E1 -24801.045,E2 -24801.045} C_VEL
LIN {X 0,Y 161.693,Z 222.164,A -85,B 0,C 180,E1 -24804.481,E2 -24804.481} C_VEL
LIN {X 0,Y 156.622,Z 214.697,A -85,B 0,C 180,E1 -24807.817,E2 -24807.817} C_VEL
LIN {X 0,Y 153.297,Z 210.161,A -85,B 0,C 180,E1 -24810.286,E2 -24810.286} C_VEL
LIN {X 0,Y 150.639,Z 206.687,A -85,B 0,C 180,E1 -24812.474,E2 -24812.474} C_VEL
LIN {X 0,Y 149.857,Z 205.631,A -85,B 0,C 180,E1 -24813.169,E2 -24813.169} C_VEL
LIN {X 0,Y 147.245,Z 202.814,A -85,B 0,C 180,E1 -24815.598,E2 -24815.598} C_VEL
LIN {X 0,Y 146,Z 200.638,A -85,B 0,C 180,E1 -24816.978,E2 -24816.978} C_VEL
LIN {X 0,Y 143.516,Z 198.655,A -85,B 0,C 180,E1 -24819.743,E2 -24819.743} C_VEL
LIN {X 0,Y 141.844,Z 195.765,A -85,B 0,C 180,E1 -24822.149,E2 -24822.149} C_VEL
LIN {X 0,Y 141.045,Z 194.888,A -85,B 0,C 180,E1 -24823.352,E2 -24823.352} C_VEL
LIN {X 0,Y 138.489,Z 193.103,A -85,B 0,C 180,E1 -24827.855,E2 -24827.855} C_VEL
LIN {X 0,Y 136.719,Z 189.805,A -85,B 0,C 180,E1 -24834.101,E2 -24834.101} C_VEL
LIN {X 0,Y 137.029,Z 189.023,A -85,B 0,C 180,E1 -24839.267,E2 -24839.267} C_VEL
LIN {X 0,Y 136.871,Z 189.121,A -85,B 0,C 180,E1 -24842.209,E2 -24842.209} C_VEL
LIN {X 0,Y 136.796,Z 190.125,A -85,B 0,C 180,E1 -24846.269,E2 -24846.269} C_VEL
LIN {X 0,Y 139.728,Z 194.225,A -85,B 0,C 180,E1 -24854.195,E2 -24854.195} C_VEL
LIN {X 0,Y 141.634,Z 195.365,A -85,B 0,C 180,E1 -24857.137,E2 -24857.137} C_VEL
LIN {X 0,Y 143.374,Z 198.483,A -85,B 0,C 180,E1 -24859.696,E2 -24859.696} C_VEL
LIN {X 0,Y 146.227,Z 200.974,A -85,B 0,C 180,E1 -24862.894,E2 -24862.894} C_VEL
LIN {X 0,Y 148.293,Z 204.202,A -85,B 0,C 180,E1 -24865.062,E2 -24865.062} C_VEL
LIN {X 0,Y 150.474,Z 206.345,A -85,B 0,C 180,E1 -24866.989,E2 -24866.989} C_VEL
LIN {X 0,Y 153.048,Z 209.935,A -85,B 0,C 180,E1 -24869.148,E2 -24869.148} C_VEL
LIN {X 0,Y 154.447,Z 211.799,A -85,B 0,C 180,E1 -24870.227,E2 -24870.227} C_VEL
LIN {X 0,Y 157.839,Z 216.537,A -85,B 0,C 180,E1 -24872.654,E2 -24872.654} C_VEL
LIN {X 0,Y 159.85,Z 219.793,A -85,B 0,C 180,E1 -24874.01,E2 -24874.01} C_VEL
LIN {X 0,Y 163.928,Z 227.35,A -85,B 0,C 180,E1 -24876.6,E2 -24876.6} C_VEL
LIN {X 0,Y 169.621,Z 239.495,A -85,B 0,C 180,E1 -24879.888,E2 -24879.888} C_VEL
LIN {X 0,Y 174.136,Z 251.395,A -85,B 0,C 180,E1 -24882.339,E2 -24882.339} C_VEL
LIN {X 0,Y 175.074,Z 254.23,A -85,B 0,C 180,E1 -24882.839,E2 -24882.839} C_VEL
LIN {X 0,Y 175.13,Z 258.15,A -85,B 0,C 180,E1 -24883.089,E2 -24883.089} C_VEL
LIN {X 0,Y 172.666,Z 291.872,A -85,B 0,C 180,E1 -24884.328,E2 -24884.328} C_VEL
LIN {X 0,Y 170.943,Z 304.296,A -85,B 0,C 180,E1 -24885.082,E2 -24885.082} C_VEL
LIN {X 0,Y 167.913,Z 317.875,A -85,B 0,C 180,E1 -24886.322,E2 -24886.322} C_VEL
LIN {X 0,Y 165.212,Z 327.385,A -85,B 0,C 180,E1 -24887.522,E2 -24887.522} C_VEL
LIN {X 0,Y 162.152,Z 336.657,A -85,B 0,C 180,E1 -24889.039,E2 -24889.039} C_VEL
LIN {X 0,Y 158.678,Z 345.596,A -85,B 0,C 180,E1 -24890.866,E2 -24890.866} C_VEL
LIN {X 0,Y 154.919,Z 354.118,A -85,B 0,C 180,E1 -24893.052,E2 -24893.052} C_VEL
LIN {X 0,Y 151.434,Z 361.333,A -85,B 0,C 180,E1 -24895.353,E2 -24895.353} C_VEL
LIN {X 0,Y 148.279,Z 367.532,A -85,B 0,C 180,E1 -24897.777,E2 -24897.777} C_VEL
LIN {X 0,Y 144.735,Z 374.068,A -85,B 0,C 180,E1 -24900.95,E2 -24900.95} C_VEL
LIN {X 0,Y 142.345,Z 378.573,A -85,B 0,C 180,E1 -24903.618,E2 -24903.618} C_VEL
LIN {X 0,Y 139.066,Z 384.064,A -85,B 0,C 180,E1 -24907.727,E2 -24907.727} C_VEL
LIN {X 0,Y 136.484,Z 388.389,A -85,B 0,C 180,E1 -24912.004,E2 -24912.004} C_VEL
LIN {X 0,Y 135.314,Z 390.762,A -85,B 0,C 180,E1 -24914.948,E2 -24914.948} C_VEL
LIN {X 0,Y 134.43,Z 392.567,A -85,B 0,C 180,E1 -24917.929,E2 -24917.929} C_VEL
LIN {X 0,Y 133.542,Z 395.027,A -85,B 0,C 180,E1 -24923.958,E2 -24923.958} C_VEL
LIN {X 0,Y 133.414,Z 395.622,A -85,B 0,C 180,E1 -24926.98,E2 -24926.98} C_VEL
LIN {X 0,Y 133.535,Z 395.782,A -85,B 0,C 180,E1 -24930,E2 -24930} C_VEL
LIN {X 0,Y 133.4,Z 395.622,A -85,B 0,C 180,E1 -24933.02,E2 -24933.02} C_VEL
LIN {X 0,Y 133.462,Z 395.025,A -85,B 0,C 180,E1 -24936.045,E2 -24936.045} C_VEL
LIN {X 0,Y 134.378,Z 392.566,A -85,B 0,C 180,E1 -24942.075,E2 -24942.075} C_VEL
LIN {X 0,Y 135.855,Z 389.609,A -85,B 0,C 180,E1 -24946.53,E2 -24946.53} C_VEL
LIN {X 0,Y 138.12,Z 385.617,A -85,B 0,C 180,E1 -24950.866,E2 -24950.866} C_VEL
LIN {X 0,Y 141.124,Z 380.487,A -85,B 0,C 180,E1 -24955.043,E2 -24955.043} C_VEL
LIN {X 0,Y 144.184,Z 375.237,A -85,B 0,C 180,E1 -24958.368,E2 -24958.368} C_VEL
LIN {X 0,Y 147.53,Z 368.908,A -85,B 0,C 180,E1 -24961.602,E2 -24961.602} C_VEL
LIN {X 0,Y 150.625,Z 362.959,A -85,B 0,C 180,E1 -24964.049,E2 -24964.049} C_VEL
LIN {X 0,Y 154.043,Z 356.037,A -85,B 0,C 180,E1 -24966.377,E2 -24966.377} C_VEL
LIN {X 0,Y 157.685,Z 347.863,A -85,B 0,C 180,E1 -24968.607,E2 -24968.607} C_VEL
LIN {X 0,Y 161.087,Z 339.356,A -85,B 0,C 180,E1 -24970.464,E2 -24970.464} C_VEL
LIN {X 0,Y 164.154,Z 330.646,A -85,B 0,C 180,E1 -24971.986,E2 -24971.986} C_VEL
LIN {X 0,Y 167.104,Z 320.894,A -85,B 0,C 180,E1 -24973.319,E2 -24973.319} C_VEL
LIN {X 0,Y 169.304,Z 312.105,A -85,B 0,C 180,E1 -24974.259,E2 -24974.259} C_VEL
LIN {X 0,Y 171.291,Z 301.853,A -85,B 0,C 180,E1 -24975.091,E2 -24975.091} C_VEL
LIN {X 0,Y 172.634,Z 291.643,A -85,B 0,C 180,E1 -24975.694,E2 -24975.694} C_VEL
LIN {X 0,Y 172.709,Z 285.862,A -85,B 0,C 180,E1 -24976.119,E2 -24976.119} C_VEL
LIN {X 0,Y 170.105,Z 267.188,A -85,B 0,C 180,E1 -24978.185,E2 -24978.185} C_VEL
LIN {X 0,Y 170.105,Z 261.377,A -85,B 0,C 180,E1 -24978.538,E2 -24978.538} C_VEL
LIN {X 0,Y 170.311,Z 256.618,A -85,B 0,C 180,E1 -24978.756,E2 -24978.756} C_VEL
LIN {X 0,Y 165.799,Z 244.224,A -85,B 0,C 180,E1 -24981.387,E2 -24981.387} C_VEL
LIN {X 0,Y 160.354,Z 232.059,A -85,B 0,C 180,E1 -24984.786,E2 -24984.786} C_VEL
LIN {X 0,Y 155.949,Z 223.632,A -85,B 0,C 180,E1 -24987.834,E2 -24987.834} C_VEL
LIN {X 0,Y 152.979,Z 219.312,A -85,B 0,C 180,E1 -24990.028,E2 -24990.028} C_VEL
LIN {X 0,Y 150.633,Z 216.029,A -85,B 0,C 180,E1 -24991.923,E2 -24991.923} C_VEL
LIN {X 0,Y 147.798,Z 212.042,A -85,B 0,C 180,E1 -24994.474,E2 -24994.474} C_VEL
LIN {X 0,Y 145.078,Z 208.846,A -85,B 0,C 180,E1 -24997.197,E2 -24997.197} C_VEL
LIN {X 0,Y 143.981,Z 207.127,A -85,B 0,C 180,E1 -24998.475,E2 -24998.475} C_VEL
LIN {X 0,Y 141.343,Z 204.483,A -85,B 0,C 180,E1 -25001.752,E2 -25001.752} C_VEL
LIN {X 0,Y 139.98,Z 201.881,A -85,B 0,C 180,E1 -25003.968,E2 -25003.968} C_VEL
LIN {X 0,Y 137.251,Z 199.851,A -85,B 0,C 180,E1 -25009.033,E2 -25009.033} C_VEL
LIN {X 0,Y 135.51,Z 196.542,A -85,B 0,C 180,E1 -25015.537,E2 -25015.537} C_VEL
LIN {X 0,Y 135.155,Z 195.799,A -85,B 0,C 180,E1 -25019.998,E2 -25019.998} C_VEL
LIN {X 0,Y 135.568,Z 196.653,A -85,B 0,C 180,E1 -25025.204,E2 -25025.204} C_VEL
LIN {X 0,Y 138.877,Z 201.335,A -85,B 0,C 180,E1 -25034.655,E2 -25034.655} C_VEL
LIN {X 0,Y 140.214,Z 202.215,A -85,B 0,C 180,E1 -25036.796,E2 -25036.796} C_VEL
LIN {X 0,Y 142.111,Z 205.506,A -85,B 0,C 180,E1 -25039.687,E2 -25039.687} C_VEL
LIN {X 0,Y 144.471,Z 207.687,A -85,B 0,C 180,E1 -25042.46,E2 -25042.46} C_VEL
LIN {X 0,Y 146.777,Z 211.094,A -85,B 0,C 180,E1 -25044.957,E2 -25044.957} C_VEL
LIN {X 0,Y 148.302,Z 212.682,A -85,B 0,C 180,E1 -25046.376,E2 -25046.376} C_VEL
LIN {X 0,Y 151.121,Z 216.526,A -85,B 0,C 180,E1 -25048.847,E2 -25048.847} C_VEL
LIN {X 0,Y 155.309,Z 222.69,A -85,B 0,C 180,E1 -25052.09,E2 -25052.09} C_VEL
LIN {X 0,Y 159.594,Z 229.256,A -85,B 0,C 180,E1 -25054.993,E2 -25054.993} C_VEL
LIN {X 0,Y 165.247,Z 238.857,A -85,B 0,C 180,E1 -25058.386,E2 -25058.386} C_VEL
LIN {X 0,Y 170.877,Z 250.01,A -85,B 0,C 180,E1 -25061.427,E2 -25061.427} C_VEL
LIN {X 0,Y 176.178,Z 262.624,A -85,B 0,C 180,E1 -25064.088,E2 -25064.088} C_VEL
LIN {X 0,Y 183.386,Z 280.226,A -85,B 0,C 180,E1 -25067.333,E2 -25067.333} C_VEL
LIN {X 0,Y 189.107,Z 292.09,A -85,B 0,C 180,E1 -25069.833,E2 -25069.833} C_VEL
LIN {X 0,Y 194.957,Z 302.955,A -85,B 0,C 180,E1 -25072.472,E2 -25072.472} C_VEL
LIN {X 0,Y 200.114,Z 311.234,A -85,B 0,C 180,E1 -25074.738,E2 -25074.738} C_VEL
LIN {X 0,Y 206.445,Z 320.149,A -85,B 0,C 180,E1 -25077.409,E2 -25077.409} C_VEL
LIN {X 0,Y 213.158,Z 328.317,A -85,B 0,C 180,E1 -25080.064,E2 -25080.064} C_VEL
LIN {X 0,Y 222.517,Z 337.836,A -85,B 0,C 180,E1 -25083.445,E2 -25083.445} C_VEL
LIN {X 0,Y 232.096,Z 345.54,A -85,B 0,C 180,E1 -25086.453,E2 -25086.453} C_VEL
LIN {X 0,Y 244.051,Z 353.488,A -85,B 0,C 180,E1 -25089.784,E2 -25089.784} C_VEL
LIN {X 0,Y 257.124,Z 360.809,A -85,B 0,C 180,E1 -25093.066,E2 -25093.066} C_VEL
LIN {X 0,Y 268.193,Z 366.679,A -85,B 0,C 180,E1 -25095.829,E2 -25095.829} C_VEL
LIN {X 0,Y 273.737,Z 369.697,A -85,B 0,C 180,E1 -25097.318,E2 -25097.318} C_VEL
LIN {X 0,Y 279.286,Z 372.81,A -85,B 0,C 180,E1 -25098.928,E2 -25098.928} C_VEL
LIN {X 0,Y 284.873,Z 375.887,A -85,B 0,C 180,E1 -25100.684,E2 -25100.684} C_VEL
LIN {X 0,Y 288.785,Z 378.411,A -85,B 0,C 180,E1 -25102.309,E2 -25102.309} C_VEL
LIN {X 0,Y 293.063,Z 381.041,A -85,B 0,C 180,E1 -25104.496,E2 -25104.496} C_VEL
LIN {X 0,Y 295.821,Z 382.45,A -85,B 0,C 180,E1 -25106.202,E2 -25106.202} C_VEL
LIN {X 0,Y 297.149,Z 383.061,A -85,B 0,C 180,E1 -25107.289,E2 -25107.289} C_VEL
LIN {X 0,Y 298.286,Z 383.475,A -85,B 0,C 180,E1 -25108.65,E2 -25108.65} C_VEL
LIN {X 0,Y 298.856,Z 383.576,A -85,B 0,C 180,E1 -25110,E2 -25110} C_VEL
LIN {X 0,Y 298.295,Z 383.48,A -85,B 0,C 180,E1 -25111.35,E2 -25111.35} C_VEL
LIN {X 0,Y 297.182,Z 383.071,A -85,B 0,C 180,E1 -25112.711,E2 -25112.711} C_VEL
LIN {X 0,Y 295.389,Z 382.268,A -85,B 0,C 180,E1 -25114.093,E2 -25114.093} C_VEL
LIN {X 0,Y 293.093,Z 381.046,A -85,B 0,C 180,E1 -25115.504,E2 -25115.504} C_VEL
LIN {X 0,Y 290.289,Z 379.425,A -85,B 0,C 180,E1 -25116.97,E2 -25116.97} C_VEL
LIN {X 0,Y 287.026,Z 377.296,A -85,B 0,C 180,E1 -25118.448,E2 -25118.448} C_VEL
LIN {X 0,Y 284.872,Z 375.889,A -85,B 0,C 180,E1 -25119.315,E2 -25119.315} C_VEL
LIN {X 0,Y 279.282,Z 372.82,A -85,B 0,C 180,E1 -25121.068,E2 -25121.068} C_VEL
LIN {X 0,Y 270.657,Z 368.046,A -85,B 0,C 180,E1 -25123.515,E2 -25123.515} C_VEL
LIN {X 0,Y 261.072,Z 362.96,A -85,B 0,C 180,E1 -25125.949,E2 -25125.949} C_VEL
LIN {X 0,Y 248.951,Z 356.338,A -85,B 0,C 180,E1 -25128.967,E2 -25128.967} C_VEL
LIN {X 0,Y 235.764,Z 348.207,A -85,B 0,C 180,E1 -25132.471,E2 -25132.471} C_VEL
LIN {X 0,Y 224.1,Z 339.175,A -85,B 0,C 180,E1 -25136.043,E2 -25136.043} C_VEL
LIN {X 0,Y 216.386,Z 331.819,A -85,B 0,C 180,E1 -25138.728,E2 -25138.728} C_VEL
LIN {X 0,Y 208.601,Z 322.875,A -85,B 0,C 180,E1 -25141.721,E2 -25141.721} C_VEL
LIN {X 0,Y 202.206,Z 314.322,A -85,B 0,C 180,E1 -25144.366,E2 -25144.366} C_VEL
LIN {X 0,Y 195.983,Z 304.703,A -85,B 0,C 180,E1 -25147.073,E2 -25147.073} C_VEL
LIN {X 0,Y 190.14,Z 293.995,A -85,B 0,C 180,E1 -25149.713,E2 -25149.713} C_VEL
LIN {X 0,Y 184.736,Z 283.014,A -85,B 0,C 180,E1 -25152.113,E2 -25152.113} C_VEL
LIN {X 0,Y 178.005,Z 267.472,A -85,B 0,C 180,E1 -25155.031,E2 -25155.031} C_VEL
LIN {X 0,Y 172.838,Z 254.438,A -85,B 0,C 180,E1 -25157.568,E2 -25157.568} C_VEL
LIN {X 0,Y 168.62,Z 245.33,A -85,B 0,C 180,E1 -25159.759,E2 -25159.759} C_VEL
LIN {X 0,Y 164.006,Z 236.671,A -85,B 0,C 180,E1 -25162.322,E2 -25162.322} C_VEL
LIN {X 0,Y 158.497,Z 227.525,A -85,B 0,C 180,E1 -25165.719,E2 -25165.719} C_VEL
LIN {X 0,Y 153.893,Z 220.519,A -85,B 0,C 180,E1 -25168.96,E2 -25168.96} C_VEL
LIN {X 0,Y 150.651,Z 216.029,A -85,B 0,C 180,E1 -25171.531,E2 -25171.531} C_VEL
LIN {X 0,Y 147.794,Z 212.057,A -85,B 0,C 180,E1 -25174.096,E2 -25174.096} C_VEL
LIN {X 0,Y 145.148,Z 208.939,A -85,B 0,C 180,E1 -25176.741,E2 -25176.741} C_VEL
LIN {X 0,Y 144.009,Z 207.181,A -85,B 0,C 180,E1 -25178.06,E2 -25178.06} C_VEL
LIN {X 0,Y 141.489,Z 204.681,A -85,B 0,C 180,E1 -25181.165,E2 -25181.165} C_VEL
LIN {X 0,Y 139.973,Z 201.891,A -85,B 0,C 180,E1 -25183.596,E2 -25183.596} C_VEL
LIN {X 0,Y 137.349,Z 199.961,A -85,B 0,C 180,E1 -25188.418,E2 -25188.418} C_VEL
LIN {X 0,Y 135.567,Z 196.665,A -85,B 0,C 180,E1 -25194.796,E2 -25194.796} C_VEL
LIN {X 0,Y 135.158,Z 195.772,A -85,B 0,C 180,E1 -25200.002,E2 -25200.002} C_VEL
LIN {X 0,Y 135.633,Z 196.792,A -85,B 0,C 180,E1 -25205.204,E2 -25205.204} C_VEL
LIN {X 0,Y 138.682,Z 201.198,A -85,B 0,C 180,E1 -25213.93,E2 -25213.93} C_VEL
LIN {X 0,Y 140.196,Z 202.157,A -85,B 0,C 180,E1 -25216.38,E2 -25216.38} C_VEL
LIN {X 0,Y 141.865,Z 205.166,A -85,B 0,C 180,E1 -25218.974,E2 -25218.974} C_VEL
LIN {X 0,Y 144.454,Z 207.699,A -85,B 0,C 180,E1 -25222.065,E2 -25222.065} C_VEL
LIN {X 0,Y 146.766,Z 211.079,A -85,B 0,C 180,E1 -25224.566,E2 -25224.566} C_VEL
LIN {X 0,Y 148.398,Z 212.85,A -85,B 0,C 180,E1 -25226.089,E2 -25226.089} C_VEL
LIN {X 0,Y 152.167,Z 218.158,A -85,B 0,C 180,E1 -25229.333,E2 -25229.333} C_VEL
LIN {X 0,Y 155.34,Z 222.748,A -85,B 0,C 180,E1 -25231.734,E2 -25231.734} C_VEL
LIN {X 0,Y 158.704,Z 228.801,A -85,B 0,C 180,E1 -25234.112,E2 -25234.112} C_VEL
LIN {X 0,Y 163.572,Z 239.076,A -85,B 0,C 180,E1 -25237.27,E2 -25237.27} C_VEL
LIN {X 0,Y 167.451,Z 248.549,A -85,B 0,C 180,E1 -25239.595,E2 -25239.595} C_VEL
LIN {X 0,Y 170.397,Z 256.918,A -85,B 0,C 180,E1 -25241.295,E2 -25241.295} C_VEL
LIN {X 0,Y 167.808,Z 291.379,A -85,B 0,C 180,E1 -25242.575,E2 -25242.575} C_VEL
LIN {X 0,Y 166.042,Z 303.812,A -85,B 0,C 180,E1 -25243.334,E2 -25243.334} C_VEL
LIN {X 0,Y 162.861,Z 317.683,A -85,B 0,C 180,E1 -25244.6,E2 -25244.6} C_VEL
LIN {X 0,Y 160.056,Z 327.193,A -85,B 0,C 180,E1 -25245.809,E2 -25245.809} C_VEL
LIN {X 0,Y 156.851,Z 336.465,A -85,B 0,C 180,E1 -25247.336,E2 -25247.336} C_VEL
LIN {X 0,Y 153.241,Z 345.405,A -85,B 0,C 180,E1 -25249.191,E2 -25249.191} C_VEL
LIN {X 0,Y 149.301,Z 353.927,A -85,B 0,C 180,E1 -25251.413,E2 -25251.413} C_VEL
LIN {X 0,Y 145.641,Z 361.141,A -85,B 0,C 180,E1 -25253.763,E2 -25253.763} C_VEL
LIN {X 0,Y 142.308,Z 367.34,A -85,B 0,C 180,E1 -25256.249,E2 -25256.249} C_VEL
LIN {X 0,Y 138.302,Z 374.285,A -85,B 0,C 180,E1 -25259.757,E2 -25259.757} C_VEL
LIN {X 0,Y 136.015,Z 378.382,A -85,B 0,C 180,E1 -25262.288,E2 -25262.288} C_VEL
LIN {X 0,Y 132.497,Z 383.871,A -85,B 0,C 180,E1 -25266.558,E2 -25266.558} C_VEL
LIN {X 0,Y 129.717,Z 388.196,A -85,B 0,C 180,E1 -25271.03,E2 -25271.03} C_VEL
LIN {X 0,Y 128.433,Z 390.569,A -85,B 0,C 180,E1 -25274.121,E2 -25274.121} C_VEL
LIN {X 0,Y 127.459,Z 392.374,A -85,B 0,C 180,E1 -25277.258,E2 -25277.258} C_VEL
LIN {X 0,Y 126.463,Z 394.835,A -85,B 0,C 180,E1 -25283.619,E2 -25283.619} C_VEL
LIN {X 0,Y 126.317,Z 395.43,A -85,B 0,C 180,E1 -25286.811,E2 -25286.811} C_VEL
LIN {X 0,Y 126.431,Z 395.591,A -85,B 0,C 180,E1 -25290,E2 -25290} C_VEL
LIN {X 0,Y 126.305,Z 395.43,A -85,B 0,C 180,E1 -25293.19,E2 -25293.19} C_VEL
LIN {X 0,Y 126.405,Z 394.834,A -85,B 0,C 180,E1 -25296.384,E2 -25296.384} C_VEL
LIN {X 0,Y 127.418,Z 392.373,A -85,B 0,C 180,E1 -25302.746,E2 -25302.746} C_VEL
LIN {X 0,Y 129.036,Z 389.416,A -85,B 0,C 180,E1 -25307.431,E2 -25307.431} C_VEL
LIN {X 0,Y 131.486,Z 385.425,A -85,B 0,C 180,E1 -25311.972,E2 -25311.972} C_VEL
LIN {X 0,Y 134.711,Z 380.295,A -85,B 0,C 180,E1 -25316.324,E2 -25316.324} C_VEL
LIN {X 0,Y 137.939,Z 375.035,A -85,B 0,C 180,E1 -25319.785,E2 -25319.785} C_VEL
LIN {X 0,Y 141.508,Z 368.715,A -85,B 0,C 180,E1 -25323.114,E2 -25323.114} C_VEL
LIN {X 0,Y 144.786,Z 362.767,A -85,B 0,C 180,E1 -25325.625,E2 -25325.625} C_VEL
LIN {X 0,Y 148.373,Z 355.845,A -85,B 0,C 180,E1 -25328.008,E2 -25328.008} C_VEL
LIN {X 0,Y 152.185,Z 347.671,A -85,B 0,C 180,E1 -25330.28,E2 -25330.28} C_VEL
LIN {X 0,Y 155.764,Z 339.165,A -85,B 0,C 180,E1 -25332.156,E2 -25332.156} C_VEL
LIN {X 0,Y 158.956,Z 330.455,A -85,B 0,C 180,E1 -25333.696,E2 -25333.696} C_VEL
LIN {X 0,Y 162.016,Z 320.703,A -85,B 0,C 180,E1 -25335.04,E2 -25335.04} C_VEL
LIN {X 0,Y 164.306,Z 311.914,A -85,B 0,C 180,E1 -25335.982,E2 -25335.982} C_VEL
LIN {X 0,Y 166.365,Z 301.593,A -85,B 0,C 180,E1 -25336.828,E2 -25336.828} C_VEL
LIN {X 0,Y 167.781,Z 291.272,A -85,B 0,C 180,E1 -25337.434,E2 -25337.434} C_VEL
LIN {X 0,Y 170.105,Z 261.377,A -85,B 0,C 180,E1 -25338.538,E2 -25338.538} C_VEL
LIN {X 0,Y 169.885,Z 259.004,A -85,B 0,C 180,E1 -25338.77,E2 -25338.77} C_VEL
LIN {X 0,Y 168.537,Z 256.069,A -85,B 0,C 180,E1 -25339.48,E2 -25339.48} C_VEL
LIN {X 0,Y 166.615,Z 253.824,A -85,B 0,C 180,E1 -25340.402,E2 -25340.402} C_VEL
LIN {X 0,Y 162.988,Z 250.204,A -85,B 0,C 180,E1 -25342.212,E2 -25342.212} C_VEL
LIN {X 0,Y 161.393,Z 247.251,A -85,B 0,C 180,E1 -25343.156,E2 -25343.156} C_VEL
LIN {X 0,Y 156.596,Z 236.235,A -85,B 0,C 180,E1 -25346.43,E2 -25346.43} C_VEL
LIN {X 0,Y 152.863,Z 228.882,A -85,B 0,C 180,E1 -25349.236,E2 -25349.236} C_VEL
LIN {X 0,Y 148.616,Z 222.507,A -85,B 0,C 180,E1 -25352.733,E2 -25352.733} C_VEL
LIN {X 0,Y 145.776,Z 218.452,A -85,B 0,C 180,E1 -25355.428,E2 -25355.428} C_VEL
LIN {X 0,Y 142.992,Z 214.893,A -85,B 0,C 180,E1 -25358.437,E2 -25358.437} C_VEL
LIN {X 0,Y 142.089,Z 213.625,A -85,B 0,C 180,E1 -25359.546,E2 -25359.546} C_VEL
LIN {X 0,Y 139.425,Z 210.432,A -85,B 0,C 180,E1 -25363.225,E2 -25363.225} C_VEL
LIN {X 0,Y 138.574,Z 208.709,A -85,B 0,C 180,E1 -25364.745,E2 -25364.745} C_VEL
LIN {X 0,Y 136.038,Z 206.57,A -85,B 0,C 180,E1 -25369.856,E2 -25369.856} C_VEL
LIN {X 0,Y 134.585,Z 203.532,A -85,B 0,C 180,E1 -25375.881,E2 -25375.881} C_VEL
LIN {X 0,Y 134.289,Z 202.855,A -85,B 0,C 180,E1 -25379.998,E2 -25379.998} C_VEL
LIN {X 0,Y 134.682,Z 203.742,A -85,B 0,C 180,E1 -25385.144,E2 -25385.144} C_VEL
LIN {X 0,Y 137.67,Z 208.225,A -85,B 0,C 180,E1 -25394.106,E2 -25394.106} C_VEL
LIN {X 0,Y 138.771,Z 209.004,A -85,B 0,C 180,E1 -25395.983,E2 -25395.983} C_VEL
LIN {X 0,Y 140.738,Z 212.37,A -85,B 0,C 180,E1 -25399.128,E2 -25399.128} C_VEL
LIN {X 0,Y 142.709,Z 214.323,A -85,B 0,C 180,E1 -25401.579,E2 -25401.579} C_VEL
LIN {X 0,Y 145.281,Z 217.964,A -85,B 0,C 180,E1 -25404.468,E2 -25404.468} C_VEL
LIN {X 0,Y 146.498,Z 219.543,A -85,B 0,C 180,E1 -25405.679,E2 -25405.679} C_VEL
LIN {X 0,Y 149.678,Z 224.078,A -85,B 0,C 180,E1 -25408.576,E2 -25408.576} C_VEL
LIN {X 0,Y 154.074,Z 230.663,A -85,B 0,C 180,E1 -25412.041,E2 -25412.041} C_VEL
LIN {X 0,Y 160.001,Z 240.719,A -85,B 0,C 180,E1 -25416.071,E2 -25416.071} C_VEL
LIN {X 0,Y 164.275,Z 248.968,A -85,B 0,C 180,E1 -25418.655,E2 -25418.655} C_VEL
LIN {X 0,Y 168.46,Z 258.128,A -85,B 0,C 180,E1 -25421.001,E2 -25421.001} C_VEL
LIN {X 0,Y 172.469,Z 268.44,A -85,B 0,C 180,E1 -25423.142,E2 -25423.142} C_VEL
LIN {X 0,Y 178.524,Z 283.786,A -85,B 0,C 180,E1 -25426.128,E2 -25426.128} C_VEL
LIN {X 0,Y 182.811,Z 293.262,A -85,B 0,C 180,E1 -25428.248,E2 -25428.248} C_VEL
LIN {X 0,Y 187.178,Z 302.281,A -85,B 0,C 180,E1 -25430.493,E2 -25430.493} C_VEL
LIN {X 0,Y 191.642,Z 310.582,A -85,B 0,C 180,E1 -25432.774,E2 -25432.774} C_VEL
LIN {X 0,Y 197.724,Z 320.162,A -85,B 0,C 180,E1 -25435.729,E2 -25435.729} C_VEL
LIN {X 0,Y 205.192,Z 330.006,A -85,B 0,C 180,E1 -25439.086,E2 -25439.086} C_VEL
LIN {X 0,Y 213.839,Z 339.214,A -85,B 0,C 180,E1 -25442.543,E2 -25442.543} C_VEL
LIN {X 0,Y 223.322,Z 347.328,A -85,B 0,C 180,E1 -25445.87,E2 -25445.87} C_VEL
LIN {X 0,Y 236.056,Z 355.823,A -85,B 0,C 180,E1 -25449.688,E2 -25449.688} C_VEL
LIN {X 0,Y 249.556,Z 363.113,A -85,B 0,C 180,E1 -25453.234,E2 -25453.234} C_VEL
LIN {X 0,Y 260.679,Z 368.596,A -85,B 0,C 180,E1 -25456.062,E2 -25456.062} C_VEL
LIN {X 0,Y 269.175,Z 372.79,A -85,B 0,C 180,E1 -25458.371,E2 -25458.371} C_VEL
LIN {X 0,Y 275.838,Z 376.141,A -85,B 0,C 180,E1 -25460.379,E2 -25460.379} C_VEL
LIN {X 0,Y 278.646,Z 377.527,A -85,B 0,C 180,E1 -25461.296,E2 -25461.296} C_VEL
LIN {X 0,Y 283.092,Z 380.124,A -85,B 0,C 180,E1 -25463.226,E2 -25463.226} C_VEL
LIN {X 0,Y 285.25,Z 381.389,A -85,B 0,C 180,E1 -25464.344,E2 -25464.344} C_VEL
LIN {X 0,Y 288.723,Z 383.147,A -85,B 0,C 180,E1 -25466.367,E2 -25466.367} C_VEL
LIN {X 0,Y 289.815,Z 383.62,A -85,B 0,C 180,E1 -25467.22,E2 -25467.22} C_VEL
LIN {X 0,Y 291.09,Z 384.126,A -85,B 0,C 180,E1 -25468.617,E2 -25468.617} C_VEL
LIN {X 0,Y 291.774,Z 384.269,A -85,B 0,C 180,E1 -25470,E2 -25470} C_VEL
LIN {X 0,Y 291.103,Z 384.128,A -85,B 0,C 180,E1 -25471.383,E2 -25471.383} C_VEL
LIN {X 0,Y 289.846,Z 383.618,A -85,B 0,C 180,E1 -25472.78,E2 -25472.78} C_VEL
LIN {X 0,Y 287.803,Z 382.704,A -85,B 0,C 180,E1 -25474.201,E2 -25474.201} C_VEL
LIN {X 0,Y 285.277,Z 381.389,A -85,B 0,C 180,E1 -25475.655,E2 -25475.655} C_VEL
LIN {X 0,Y 282.354,Z 379.675,A -85,B 0,C 180,E1 -25477.149,E2 -25477.149} C_VEL
LIN {X 0,Y 277.559,Z 376.962,A -85,B 0,C 180,E1 -25479.072,E2 -25479.072} C_VEL
LIN {X 0,Y 271.891,Z 374.191,A -85,B 0,C 180,E1 -25480.817,E2 -25480.817} C_VEL
LIN {X 0,Y 266.283,Z 371.364,A -85,B 0,C 180,E1 -25482.44,E2 -25482.44} C_VEL
LIN {X 0,Y 258.706,Z 367.655,A -85,B 0,C 180,E1 -25484.43,E2 -25484.43} C_VEL
LIN {X 0,Y 246.809,Z 361.7,A -85,B 0,C 180,E1 -25487.463,E2 -25487.463} C_VEL
LIN {X 0,Y 232.701,Z 353.807,A -85,B 0,C 180,E1 -25491.249,E2 -25491.249} C_VEL
LIN {X 0,Y 221.623,Z 345.963,A -85,B 0,C 180,E1 -25494.7,E2 -25494.7} C_VEL
LIN {X 0,Y 211.9,Z 337.33,A -85,B 0,C 180,E1 -25498.196,E2 -25498.196} C_VEL
LIN {X 0,Y 203.611,Z 327.968,A -85,B 0,C 180,E1 -25501.633,E2 -25501.633} C_VEL
LIN {X 0,Y 195.861,Z 317.285,A -85,B 0,C 180,E1 -25505.193,E2 -25505.193} C_VEL
LIN {X 0,Y 189.729,Z 307.117,A -85,B 0,C 180,E1 -25508.218,E2 -25508.218} C_VEL
LIN {X 0,Y 183.891,Z 295.622,A -85,B 0,C 180,E1 -25511.201,E2 -25511.201} C_VEL
LIN {X 0,Y 178.821,Z 284.332,A -85,B 0,C 180,E1 -25513.768,E2 -25513.768} C_VEL
LIN {X 0,Y 172.567,Z 268.791,A -85,B 0,C 180,E1 -25516.802,E2 -25516.802} C_VEL
LIN {X 0,Y 168.665,Z 258.629,A -85,B 0,C 180,E1 -25518.886,E2 -25518.886} C_VEL
LIN {X 0,Y 164.564,Z 249.529,A -85,B 0,C 180,E1 -25521.181,E2 -25521.181} C_VEL
LIN {X 0,Y 160.394,Z 241.467,A -85,B 0,C 180,E1 -25523.68,E2 -25523.68} C_VEL
LIN {X 0,Y 155.557,Z 233.155,A -85,B 0,C 180,E1 -25526.882,E2 -25526.882} C_VEL
LIN {X 0,Y 151.343,Z 226.466,A -85,B 0,C 180,E1 -25530.055,E2 -25530.055} C_VEL
LIN {X 0,Y 148.301,Z 222.144,A -85,B 0,C 180,E1 -25532.625,E2 -25532.625} C_VEL
LIN {X 0,Y 145.607,Z 218.305,A -85,B 0,C 180,E1 -25535.21,E2 -25535.21} C_VEL
LIN {X 0,Y 142.907,Z 214.707,A -85,B 0,C 180,E1 -25538.168,E2 -25538.168} C_VEL
LIN {X 0,Y 142.22,Z 213.761,A -85,B 0,C 180,E1 -25539.008,E2 -25539.008} C_VEL
LIN {X 0,Y 139.68,Z 210.873,A -85,B 0,C 180,E1 -25542.431,E2 -25542.431} C_VEL
LIN {X 0,Y 138.682,Z 208.756,A -85,B 0,C 180,E1 -25544.195,E2 -25544.195} C_VEL
LIN {X 0,Y 136.219,Z 206.835,A -85,B 0,C 180,E1 -25548.994,E2 -25548.994} C_VEL
LIN {X 0,Y 134.637,Z 203.658,A -85,B 0,C 180,E1 -25555.136,E2 -25555.136} C_VEL
LIN {X 0,Y 134.294,Z 202.81,A -85,B 0,C 180,E1 -25560.002,E2 -25560.002} C_VEL
LIN {X 0,Y 134.697,Z 203.791,A -85,B 0,C 180,E1 -25564.865,E2 -25564.865} C_VEL
LIN {X 0,Y 137.443,Z 208.066,A -85,B 0,C 180,E1 -25573.305,E2 -25573.305} C_VEL
LIN {X 0,Y 138.798,Z 209.063,A -85,B 0,C 180,E1 -25575.653,E2 -25575.653} C_VEL
LIN {X 0,Y 140.745,Z 212.34,A -85,B 0,C 180,E1 -25578.752,E2 -25578.752} C_VEL
LIN {X 0,Y 142.72,Z 214.356,A -85,B 0,C 180,E1 -25581.215,E2 -25581.215} C_VEL
LIN {X 0,Y 145.283,Z 217.976,A -85,B 0,C 180,E1 -25584.091,E2 -25584.091} C_VEL
LIN {X 0,Y 146.496,Z 219.527,A -85,B 0,C 180,E1 -25585.296,E2 -25585.296} C_VEL
LIN {X 0,Y 149.766,Z 224.245,A -85,B 0,C 180,E1 -25588.274,E2 -25588.274} C_VEL
LIN {X 0,Y 153.254,Z 229.477,A -85,B 0,C 180,E1 -25591.06,E2 -25591.06} C_VEL
LIN {X 0,Y 157.895,Z 239.05,A -85,B 0,C 180,E1 -25594.49,E2 -25594.49} C_VEL
LIN {X 0,Y 162.607,Z 250.354,A -85,B 0,C 180,E1 -25597.627,E2 -25597.627} C_VEL
LIN {X 0,Y 165.618,Z 259.105,A -85,B 0,C 180,E1 -25599.535,E2 -25599.535} C_VEL
LIN {X 0,Y 163.069,Z 291.349,A -85,B 0,C 180,E1 -25600.745,E2 -25600.745} C_VEL
LIN {X 0,Y 161.28,Z 303.5,A -85,B 0,C 180,E1 -25601.493,E2 -25601.493} C_VEL
LIN {X 0,Y 157.968,Z 317.492,A -85,B 0,C 180,E1 -25602.771,E2 -25602.771} C_VEL
LIN {X 0,Y 155.045,Z 327.002,A -85,B 0,C 180,E1 -25603.98,E2 -25603.98} C_VEL
LIN {X 0,Y 151.706,Z 336.274,A -85,B 0,C 180,E1 -25605.518,E2 -25605.518} C_VEL
LIN {X 0,Y 147.939,Z 345.213,A -85,B 0,C 180,E1 -25607.394,E2 -25607.394} C_VEL
LIN {X 0,Y 143.801,Z 353.734,A -85,B 0,C 180,E1 -25609.642,E2 -25609.642} C_VEL
LIN {X 0,Y 139.974,Z 360.949,A -85,B 0,C 180,E1 -25612.044,E2 -25612.044} C_VEL
LIN {X 0,Y 136.424,Z 367.147,A -85,B 0,C 180,E1 -25614.581,E2 -25614.581} C_VEL
LIN {X 0,Y 132.439,Z 373.683,A -85,B 0,C 180,E1 -25617.951,E2 -25617.951} C_VEL
LIN {X 0,Y 129.748,Z 378.189,A -85,B 0,C 180,E1 -25620.824,E2 -25620.824} C_VEL
LIN {X 0,Y 125.99,Z 383.679,A -85,B 0,C 180,E1 -25625.269,E2 -25625.269} C_VEL
LIN {X 0,Y 122.998,Z 388.004,A -85,B 0,C 180,E1 -25629.951,E2 -25629.951} C_VEL
LIN {X 0,Y 121.572,Z 390.376,A -85,B 0,C 180,E1 -25633.199,E2 -25633.199} C_VEL
LIN {X 0,Y 120.518,Z 392.182,A -85,B 0,C 180,E1 -25636.511,E2 -25636.511} C_VEL
LIN {X 0,Y 119.392,Z 394.643,A -85,B 0,C 180,E1 -25643.239,E2 -25643.239} C_VEL
LIN {X 0,Y 119.231,Z 395.239,A -85,B 0,C 180,E1 -25646.621,E2 -25646.621} C_VEL
LIN {X 0,Y 119.337,Z 395.399,A -85,B 0,C 180,E1 -25650,E2 -25650} C_VEL
LIN {X 0,Y 119.221,Z 395.238,A -85,B 0,C 180,E1 -25653.379,E2 -25653.379} C_VEL
LIN {X 0,Y 119.326,Z 394.641,A -85,B 0,C 180,E1 -25656.765,E2 -25656.765} C_VEL
LIN {X 0,Y 120.485,Z 392.181,A -85,B 0,C 180,E1 -25663.493,E2 -25663.493} C_VEL
LIN {X 0,Y 122.234,Z 389.223,A -85,B 0,C 180,E1 -25668.435,E2 -25668.435} C_VEL
LIN {X 0,Y 124.91,Z 385.233,A -85,B 0,C 180,E1 -25673.194,E2 -25673.194} C_VEL
LIN {X 0,Y 128.377,Z 380.103,A -85,B 0,C 180,E1 -25677.731,E2 -25677.731} C_VEL
LIN {X 0,Y 132.215,Z 374.173,A -85,B 0,C 180,E1 -25681.732,E2 -25681.732} C_VEL
LIN {X 0,Y 136.433,Z 367.147,A -85,B 0,C 180,E1 -25685.416,E2 -25685.416} C_VEL
LIN {X 0,Y 141.86,Z 357.57,A -85,B 0,C 180,E1 -25689.172,E2 -25689.172} C_VEL
LIN {X 0,Y 146.331,Z 348.613,A -85,B 0,C 180,E1 -25691.788,E2 -25691.788} C_VEL
LIN {X 0,Y 150.009,Z 340.323,A -85,B 0,C 180,E1 -25693.712,E2 -25693.712} C_VEL
LIN {X 0,Y 153.913,Z 330.264,A -85,B 0,C 180,E1 -25695.518,E2 -25695.518} C_VEL
LIN {X 0,Y 157.082,Z 320.511,A -85,B 0,C 180,E1 -25696.872,E2 -25696.872} C_VEL
LIN {X 0,Y 159.465,Z 311.723,A -85,B 0,C 180,E1 -25697.813,E2 -25697.813} C_VEL
LIN {X 0,Y 161.678,Z 300.966,A -85,B 0,C 180,E1 -25698.688,E2 -25698.688} C_VEL
LIN {X 0,Y 163.066,Z 291.081,A -85,B 0,C 180,E1 -25699.27,E2 -25699.27} C_VEL
LIN {X 0,Y 165.622,Z 259.07,A -85,B 0,C 180,E1 -25700.466,E2 -25700.466} C_VEL
LIN {X 0,Y 161.646,Z 247.869,A -85,B 0,C 180,E1 -25702.993,E2 -25702.993} C_VEL
LIN {X 0,Y 161.393,Z 247.251,A -85,B 0,C 180,E1 -25703.156,E2 -25703.156} C_VEL
LIN {X 0,Y 160.126,Z 244.346,A -85,B 0,C 180,E1 -25703.977,E2 -25703.977} C_VEL
LIN {X 0,Y 157.705,Z 240.883,A -85,B 0,C 180,E1 -25705.466,E2 -25705.466} C_VEL
LIN {X 0,Y 153.152,Z 236.636,A -85,B 0,C 180,E1 -25708.374,E2 -25708.374} C_VEL
LIN {X 0,Y 149.677,Z 233.415,A -85,B 0,C 180,E1 -25710.895,E2 -25710.895} C_VEL
LIN {X 0,Y 148.167,Z 231.478,A -85,B 0,C 180,E1 -25712.148,E2 -25712.148} C_VEL
LIN {X 0,Y 145.926,Z 228.111,A -85,B 0,C 180,E1 -25714.216,E2 -25714.216} C_VEL
LIN {X 0,Y 143.636,Z 224.697,A -85,B 0,C 180,E1 -25716.573,E2 -25716.573} C_VEL
LIN {X 0,Y 140.411,Z 220.236,A -85,B 0,C 180,E1 -25720.442,E2 -25720.442} C_VEL
LIN {X 0,Y 137.75,Z 216.666,A -85,B 0,C 180,E1 -25724.462,E2 -25724.462} C_VEL
LIN {X 0,Y 137.195,Z 215.517,A -85,B 0,C 180,E1 -25725.537,E2 -25725.537} C_VEL
LIN {X 0,Y 134.636,Z 212.998,A -85,B 0,C 180,E1 -25731.367,E2 -25731.367} C_VEL
LIN {X 0,Y 133.642,Z 210.473,A -85,B 0,C 180,E1 -25736.418,E2 -25736.418} C_VEL
LIN {X 0,Y 133.425,Z 209.887,A -85,B 0,C 180,E1 -25739.998,E2 -25739.998} C_VEL
LIN {X 0,Y 133.765,Z 210.786,A -85,B 0,C 180,E1 -25744.896,E2 -25744.896} C_VEL
LIN {X 0,Y 136.402,Z 215.057,A -85,B 0,C 180,E1 -25753.405,E2 -25753.405} C_VEL
LIN {X 0,Y 137.382,Z 215.824,A -85,B 0,C 180,E1 -25755.198,E2 -25755.198} C_VEL
LIN {X 0,Y 139.652,Z 219.517,A -85,B 0,C 180,E1 -25758.939,E2 -25758.939} C_VEL
LIN {X 0,Y 141.051,Z 221.039,A -85,B 0,C 180,E1 -25760.764,E2 -25760.764} C_VEL
LIN {X 0,Y 143.794,Z 224.857,A -85,B 0,C 180,E1 -25763.969,E2 -25763.969} C_VEL
LIN {X 0,Y 147.411,Z 230.31,A -85,B 0,C 180,E1 -25767.554,E2 -25767.554} C_VEL
LIN {X 0,Y 150.812,Z 235.614,A -85,B 0,C 180,E1 -25770.448,E2 -25770.448} C_VEL
LIN {X 0,Y 155.658,Z 243.991,A -85,B 0,C 180,E1 -25774.064,E2 -25774.064} C_VEL
LIN {X 0,Y 160.181,Z 252.812,A -85,B 0,C 180,E1 -25777.055,E2 -25777.055} C_VEL
LIN {X 0,Y 164.252,Z 261.938,A -85,B 0,C 180,E1 -25779.529,E2 -25779.529} C_VEL
LIN {X 0,Y 168.234,Z 272.639,A -85,B 0,C 180,E1 -25781.834,E2 -25781.834} C_VEL
LIN {X 0,Y 173.866,Z 287.643,A -85,B 0,C 180,E1 -25784.918,E2 -25784.918} C_VEL
LIN {X 0,Y 179.327,Z 300.727,A -85,B 0,C 180,E1 -25788.125,E2 -25788.125} C_VEL
LIN {X 0,Y 184.284,Z 311.145,A -85,B 0,C 180,E1 -25791.073,E2 -25791.073} C_VEL
LIN {X 0,Y 189.273,Z 319.904,A -85,B 0,C 180,E1 -25793.86,E2 -25793.86} C_VEL
LIN {X 0,Y 195.248,Z 328.761,A -85,B 0,C 180,E1 -25796.965,E2 -25796.965} C_VEL
LIN {X 0,Y 202.309,Z 337.388,A -85,B 0,C 180,E1 -25800.279,E2 -25800.279} C_VEL
LIN {X 0,Y 211.196,Z 346.14,A -85,B 0,C 180,E1 -25803.957,E2 -25803.957} C_VEL
LIN {X 0,Y 220.847,Z 353.478,A -85,B 0,C 180,E1 -25807.346,E2 -25807.346} C_VEL
LIN {X 0,Y 233.813,Z 361.22,A -85,B 0,C 180,E1 -25811.23,E2 -25811.23} C_VEL
LIN {X 0,Y 247.536,Z 367.867,A -85,B 0,C 180,E1 -25814.863,E2 -25814.863} C_VEL
LIN {X 0,Y 258.831,Z 372.905,A -85,B 0,C 180,E1 -25817.818,E2 -25817.818} C_VEL
LIN {X 0,Y 267.04,Z 376.644,A -85,B 0,C 180,E1 -25820.212,E2 -25820.212} C_VEL
LIN {X 0,Y 270.233,Z 378.058,A -85,B 0,C 180,E1 -25821.211,E2 -25821.211} C_VEL
LIN {X 0,Y 274.139,Z 379.898,A -85,B 0,C 180,E1 -25822.635,E2 -25822.635} C_VEL
LIN {X 0,Y 277.363,Z 381.604,A -85,B 0,C 180,E1 -25824.183,E2 -25824.183} C_VEL
LIN {X 0,Y 281.617,Z 383.53,A -85,B 0,C 180,E1 -25826.581,E2 -25826.581} C_VEL
LIN {X 0,Y 283.855,Z 384.397,A -85,B 0,C 180,E1 -25828.581,E2 -25828.581} C_VEL
LIN {X 0,Y 284.64,Z 384.58,A -85,B 0,C 180,E1 -25830,E2 -25830} C_VEL
LIN {X 0,Y 283.871,Z 384.396,A -85,B 0,C 180,E1 -25831.419,E2 -25831.419} C_VEL
LIN {X 0,Y 282.429,Z 383.839,A -85,B 0,C 180,E1 -25832.853,E2 -25832.853} C_VEL
LIN {X 0,Y 280.091,Z 382.911,A -85,B 0,C 180,E1 -25834.317,E2 -25834.317} C_VEL
LIN {X 0,Y 275.91,Z 380.786,A -85,B 0,C 180,E1 -25836.589,E2 -25836.589} C_VEL
LIN {X 0,Y 274.128,Z 379.899,A -85,B 0,C 180,E1 -25837.365,E2 -25837.365} C_VEL
LIN {X 0,Y 269.594,Z 377.773,A -85,B 0,C 180,E1 -25838.999,E2 -25838.999} C_VEL
LIN {X 0,Y 261.327,Z 374.064,A -85,B 0,C 180,E1 -25841.474,E2 -25841.474} C_VEL
LIN {X 0,Y 253.138,Z 370.424,A -85,B 0,C 180,E1 -25843.662,E2 -25843.662} C_VEL
LIN {X 0,Y 244.741,Z 366.606,A -85,B 0,C 180,E1 -25845.852,E2 -25845.852} C_VEL
LIN {X 0,Y 230.996,Z 359.704,A -85,B 0,C 180,E1 -25849.552,E2 -25849.552} C_VEL
LIN {X 0,Y 219.126,Z 352.301,A -85,B 0,C 180,E1 -25853.224,E2 -25853.224} C_VEL
LIN {X 0,Y 208.245,Z 343.572,A -85,B 0,C 180,E1 -25857.19,E2 -25857.19} C_VEL
LIN {X 0,Y 199.623,Z 334.346,A -85,B 0,C 180,E1 -25860.941,E2 -25860.941} C_VEL
LIN {X 0,Y 192.509,Z 324.915,A -85,B 0,C 180,E1 -25864.428,E2 -25864.428} C_VEL
LIN {X 0,Y 186.473,Z 315.186,A -85,B 0,C 180,E1 -25867.679,E2 -25867.679} C_VEL
LIN {X 0,Y 182.002,Z 306.37,A -85,B 0,C 180,E1 -25870.305,E2 -25870.305} C_VEL
LIN {X 0,Y 177.338,Z 296.058,A -85,B 0,C 180,E1 -25873.058,E2 -25873.058} C_VEL
LIN {X 0,Y 173.073,Z 285.539,A -85,B 0,C 180,E1 -25875.537,E2 -25875.537} C_VEL
LIN {X 0,Y 168.079,Z 272.199,A -85,B 0,C 180,E1 -25878.253,E2 -25878.253} C_VEL
LIN {X 0,Y 164.023,Z 261.428,A -85,B 0,C 180,E1 -25880.603,E2 -25880.603} C_VEL
LIN {X 0,Y 160.267,Z 252.997,A -85,B 0,C 180,E1 -25882.891,E2 -25882.891} C_VEL
LIN {X 0,Y 155.966,Z 244.583,A -85,B 0,C 180,E1 -25885.72,E2 -25885.72} C_VEL
LIN {X 0,Y 151.197,Z 236.18,A -85,B 0,C 180,E1 -25889.251,E2 -25889.251} C_VEL
LIN {X 0,Y 146.439,Z 228.748,A -85,B 0,C 180,E1 -25893.359,E2 -25893.359} C_VEL
LIN {X 0,Y 143.478,Z 224.533,A -85,B 0,C 180,E1 -25896.358,E2 -25896.358} C_VEL
LIN {X 0,Y 140.516,Z 220.321,A -85,B 0,C 180,E1 -25899.932,E2 -25899.932} C_VEL
LIN {X 0,Y 138.044,Z 217.231,A -85,B 0,C 180,E1 -25903.551,E2 -25903.551} C_VEL
LIN {X 0,Y 137.192,Z 215.527,A -85,B 0,C 180,E1 -25905.161,E2 -25905.161} C_VEL
LIN {X 0,Y 134.943,Z 213.431,A -85,B 0,C 180,E1 -25910.05,E2 -25910.05} C_VEL
LIN {X 0,Y 133.665,Z 210.522,A -85,B 0,C 180,E1 -25915.856,E2 -25915.856} C_VEL
LIN {X 0,Y 133.427,Z 209.871,A -85,B 0,C 180,E1 -25920.002,E2 -25920.002} C_VEL
LIN {X 0,Y 133.765,Z 210.796,A -85,B 0,C 180,E1 -25924.522,E2 -25924.522} C_VEL
LIN {X 0,Y 136.404,Z 215.058,A -85,B 0,C 180,E1 -25933.029,E2 -25933.029} C_VEL
LIN {X 0,Y 137.384,Z 215.818,A -85,B 0,C 180,E1 -25934.821,E2 -25934.821} C_VEL
LIN {X 0,Y 139.509,Z 219.319,A -85,B 0,C 180,E1 -25938.354,E2 -25938.354} C_VEL
LIN {X 0,Y 141.071,Z 221.086,A -85,B 0,C 180,E1 -25940.411,E2 -25940.411} C_VEL
LIN {X 0,Y 143.795,Z 224.853,A -85,B 0,C 180,E1 -25943.59,E2 -25943.59} C_VEL
LIN {X 0,Y 147.367,Z 230.237,A -85,B 0,C 180,E1 -25947.133,E2 -25947.133} C_VEL
LIN {X 0,Y 150.482,Z 235.155,A -85,B 0,C 180,E1 -25949.81,E2 -25949.81} C_VEL
LIN {X 0,Y 154.459,Z 243.779,A -85,B 0,C 180,E1 -25952.998,E2 -25952.998} C_VEL
LIN {X 0,Y 158.704,Z 254.387,A -85,B 0,C 180,E1 -25956.076,E2 -25956.076} C_VEL
LIN {X 0,Y 161.002,Z 261.317,A -85,B 0,C 180,E1 -25957.672,E2 -25957.672} C_VEL
LIN {X 0,Y 158.504,Z 291.4,A -85,B 0,C 180,E1 -25958.814,E2 -25958.814} C_VEL
LIN {X 0,Y 156.454,Z 304.494,A -85,B 0,C 180,E1 -25959.628,E2 -25959.628} C_VEL
LIN {X 0,Y 153.239,Z 317.301,A -85,B 0,C 180,E1 -25960.823,E2 -25960.823} C_VEL
LIN {X 0,Y 150.199,Z 326.81,A -85,B 0,C 180,E1 -25962.029,E2 -25962.029} C_VEL
LIN {X 0,Y 146.726,Z 336.082,A -85,B 0,C 180,E1 -25963.576,E2 -25963.576} C_VEL
LIN {X 0,Y 142.778,Z 345.021,A -85,B 0,C 180,E1 -25965.458,E2 -25965.458} C_VEL
LIN {X 0,Y 138.449,Z 353.542,A -85,B 0,C 180,E1 -25967.732,E2 -25967.732} C_VEL
LIN {X 0,Y 134.426,Z 360.757,A -85,B 0,C 180,E1 -25970.175,E2 -25970.175} C_VEL
LIN {X 0,Y 130.686,Z 366.955,A -85,B 0,C 180,E1 -25972.772,E2 -25972.772} C_VEL
LIN {X 0,Y 126.44,Z 373.49,A -85,B 0,C 180,E1 -25976.232,E2 -25976.232} C_VEL
LIN {X 0,Y 123.549,Z 377.996,A -85,B 0,C 180,E1 -25979.206,E2 -25979.206} C_VEL
LIN {X 0,Y 119.541,Z 383.486,A -85,B 0,C 180,E1 -25983.837,E2 -25983.837} C_VEL
LIN {X 0,Y 116.334,Z 387.812,A -85,B 0,C 180,E1 -25988.748,E2 -25988.748} C_VEL
LIN {X 0,Y 114.746,Z 390.184,A -85,B 0,C 180,E1 -25992.167,E2 -25992.167} C_VEL
LIN {X 0,Y 113.607,Z 391.99,A -85,B 0,C 180,E1 -25995.674,E2 -25995.674} C_VEL
